// TIA Portal V21 program export: 7 tag tables, 1 data types, 19 data blocks, 22 code blocks (in call order from the OBs), 253 instance data blocks

VAR_GLOBAL   // PLC tag table "ALARM BIT"
   "DOOR1 CLOSE PB BIT" AT %M145.0 : Bool;
   "PV BOILER TEMP" AT %MD146 : Real;
   "SET BOILER BIT" AT %M145.1 : Bool;
   "PLANT STEAM LOW BIT" AT %M145.2 : Bool;
   "PURE STEAM LOW BIT" AT %M145.3 : Bool;
   "COOLING WATER LOW BIT" AT %M145.4 : Bool;
   "DOOR1 SAFETY SENSOR BIT" AT %M145.5 : Bool;
   "DOOR2 SAFETY SENSOR BIT" AT %M145.6 : Bool;
   "BOILER WATER OK BIT" AT %M145.7 : Bool;
   "RESET C21" AT %M152.2 : Bool;
   "MAN BOILER INLET VAL" AT %M152.3 : Bool;
   RESET_c22 AT %M152.4 : Bool;
   PULSE63 AT %M152.5 : Bool;
   PULSE64 AT %M152.6 : Bool;
   "door2 allow" AT %M152.7 : Bool;
   Cham_exh_val_bit AT %M160.0 : Bool;
   pulse65 AT %M160.1 : Bool;
   "abort standard" AT %M160.2 : Bool;
   PULSE66 AT %M154.0 : Bool;
END_VAR

VAR_GLOBAL   // PLC tag table "ANALOG"
   "DOOR1 PRESSURE" AT %IW120 : Int;
   "DOOR2 PRESSURE" AT %IW122 : Int;
   "JACKET PRESSURE" AT %IW124 : Int;
   "CHAMBER PRESSURE" AT %IW126 : Int;
END_VAR

VAR_GLOBAL   // PLC tag table "BIT"
END_VAR

VAR_GLOBAL   // PLC tag table "DI"
   "EMG SWITCH" AT %I0.0 : Bool;
   "RESET PB" AT %I0.1 : Bool;
   "VACUUM PUMP TRIP" AT %I0.2 : Bool;
   "DOOR1 OPEN LMT" AT %I0.3 : Bool;
   "DOOR1 CLOSE LMT" AT %I0.4 : Bool;
   "DOOR2 OPEN LMT" AT %I0.5 : Bool;
   "DOOR2 CLOSE LMT" AT %I0.6 : Bool;
   "DOOR2 CLOSE PB" AT %I0.7 : Bool;
   "DOOR2 OPEN PB" AT %I1.0 : Bool;
   "DOOR1 CLOSE PB" AT %I1.1 : Bool;
   "DOOR1 OPEN PB" AT %I1.2 : Bool;
   "AIR PREESURE SWS" AT %I1.3 : Bool;
   "plant steam low" AT %I1.4 : Bool;
   "pure steam low" AT %I1.5 : Bool;
   "cooling wtr low" AT %I2.0 : Bool;
   SPP AT %I2.1 : Bool;
   "DOOR1 CURTAIN SENSOR" AT %I2.2 : Bool;
   "DOOR2 CURTAIN SENSOR" AT %I2.3 : Bool;
   "BOILER WATER LEVEL OK" AT %I2.4 : Bool;
   "DRUM VFD TRIP" AT %I10.2 : Bool;
   "CRC PUMP TRIP" AT %I10.4 : Bool;
END_VAR

VAR_GLOBAL   // PLC tag table "DO"
   "VCC PUMP" AT %Q0.0 : Bool;   // VCC PUMP
   "DOOR1 GASKET" AT %Q0.1 : Bool;   // DOOR1 GASKET
   "DOOR1 VCC" AT %Q0.2 : Bool;   // DOOR1 VCC
   "DOOR2 GASKET" AT %Q0.3 : Bool;   // DOOR2 GASKET
   "DOOR2 VCC" AT %Q0.4 : Bool;   // DOOR2 VCC
   "JACKET STEAM VAL" AT %Q0.5 : Bool;   // JACKET STEAM VAL
   "JACKET STEAM OUT" AT %Q0.6 : Bool;
   "CHAMBER STEAM VAL" AT %Q0.7 : Bool;   // CHAMBER STEAM VAL
   "CHAMBER STEAM SMALL" AT %Q1.0 : Bool;   // DOOR2 INTERLOCK VAL
   "CHAMBER EXHAUST VAL" AT %Q1.1 : Bool;   // CHAMBER EXHAUST VAL
   "DRAIN VAL" AT %Q2.0 : Bool;   // DRAIN VAL
   "CHAMBER VACCUM VAL" AT %Q2.1 : Bool;
   "CHAMBER VENT VAL" AT %Q2.2 : Bool;   // CHAMBER VENT VAL
   "DOOR1 OPEN VAL" AT %Q2.3 : Bool;   // DOOR1 OPEN VAL
   "DOOR1 CLOSE VAL" AT %Q2.4 : Bool;   // DOOR1 CLOSE VAL
   "DOOR2 OPEN VAL" AT %Q2.5 : Bool;   // DOOR2 OPEN VAL
   "DOOR2 CLOSE VAL" AT %Q2.6 : Bool;   // DOOR2 CLOSE VAL
   "PROCESS ON IND" AT %Q2.7 : Bool;   // WFI VAL
   "door1 precondition lamp" AT %Q3.0 : Bool;
   "door2 precondition lamp" AT %Q3.1 : Bool;
   "DOOR1 OPEN LAMP" AT %Q3.2 : Bool;   // PWD VAL
   "DOOR2 OPEN LAMP" AT %Q3.3 : Bool;   // PWD CRC VAL
   HOOTER AT %Q3.4 : Bool;   // HOOTER
   "CHAMBER CONDENSOR VAL" AT %Q3.5 : Bool;   // CHAMBER CONDENSOR VAL
   "BOILER HEATER" AT %Q3.6 : Bool;   // BOILER HEATER
   "CRC MOTOR" AT %Q10.2 : Bool;   // CRC MOTOR
   "DETERGENT DSG VAL" AT %Q12.2 : Bool;   // DETERGENT DSG VAL
   "SILICON DSG VAL" AT %Q12.3 : Bool;   // SILICON DSG VAL
   "CHAMBER AIR VENT FAST" AT %Q18.6 : Bool;   // DOOR1 INTERLOCK VAL
END_VAR

VAR_GLOBAL   // PLC tag table "Default tag table"
   "REC DOOR1 PRESSURE" AT %QW150 : Int;
   "REC DOOR2 PRESSURE" AT %QW152 : Int;
   "REC CHAMBER PRESSURE" AT %QW154 : Int;
   "REC JACKET PRESSURE" AT %QW156 : Int;
   "REC DRUM SPEED" AT %QW158 : Int;
   "PRINT START" AT %M0.0 : Bool;
   TRIGGER AT %M0.1 : Bool;
   LENGTH AT %MW2 : Int;
   "NOT" AT %M0.2 : Bool;
   HIT AT %M0.3 : Bool;
   "START PV" AT %M0.4 : Bool;
   Clock_Byte AT %MB500 : Byte;
   Clock_10Hz AT %M500.0 : Bool;
   Clock_5Hz AT %M500.1 : Bool;
   "Clock_2.5Hz" AT %M500.2 : Bool;
   Clock_2Hz AT %M500.3 : Bool;
   "Clock_1.25Hz" AT %M500.4 : Bool;
   Clock_1Hz AT %M500.5 : Bool;
   "Clock_0.625Hz" AT %M500.6 : Bool;
   "Clock_0.5Hz" AT %M500.7 : Bool;
   System_Byte AT %MB1 : Byte;
   FirstScan AT %M1.0 : Bool;
   DiagStatusUpdate AT %M1.1 : Bool;
   AlwaysTRUE AT %M1.2 : Bool;
   AlwaysFALSE AT %M1.3 : Bool;
   AHJGSJH AT %MB4 : Byte;
   JGJH AT %MB5 : Byte;
   GET_DAY AT %MB180 : Byte;
   GET_MONTH AT %MB181 : Byte;
   GET_YEAR AT %MB182 : Byte;
   DAY AT %MW32 : Int;
   MONTH AT %MW44 : Int;
   YEAR AT %MW10 : Int;
   GET_HOUR AT %MB183 : Byte;
   GET_MINUTE AT %MB184 : Byte;
   GET_SECOND AT %MB185 : Byte;
   HOUR AT %MW40 : Int;
   MINUTE AT %MW42 : Int;
   SECOND AT %MW12 : Int;
   "NILESH BHAU" AT %MB6 : Byte;
   GET_CONTROL_TEMP AT %MD1400 : Real;
   "SP_CONTROL TEMP" AT %MD60 : Real;
   GET_CONVEYOR_SPEED AT %MD1404 : Real;
   SP_CONVEYOR_SPEED AT %MD64 : Real;
   "DRY ZONE REAL" AT %MD16 : Real;
   "GET_CONVEYOR ON TEMP" AT %MD1408 : Real;
   SP_CONVEYOR_ON_TEMP AT %MD68 : Real;
   "GET_CONVEYOR OFF TEMP" AT %MD1412 : Real;
   SP_CONVEYOR_OFF_TEMP AT %MD72 : Real;
   GET_DZ_PV AT %MD1416 : Real;
   DZ_PV AT %MD20 : Real;
   GET_MHZ_PV AT %MD1420 : Real;
   MHZ_PV AT %MD76 : Real;
   GET_STR_IN_PV AT %MD1424 : Real;
   STR_IN_PV AT %MD24 : Real;
   GET_STR_OUT_PV AT %MD1428 : Real;
   STR_OUT_PV AT %MD80 : Real;
   GET_CLZ_UP_PV AT %MD1432 : Real;
   CLZ_UP_PV AT %MD84 : Real;
   GET_CLZ_DWN_PV AT %MD1436 : Real;
   CLZ_DWN_PV AT %MD28 : Real;
   "GET_CONVEYOR SPEED_PV" AT %MD1440 : Real;
   "CONVEYOR SPEED_PV" AT %MD36 : Real;
   KJAHKJH AT %MD46 : Real;
   GET_MODE AT %MB197 : Byte;
   MODE AT %MW14 : Int;
   GET_PROCESS_HOUR AT %MB198 : Byte;
   PROCESS_HOUR AT %MW50 : Int;
   GET_PROCESS_MINUTE AT %MB199 : Byte;
   PROCESS_MINUTE AT %MW52 : Int;
   GET_PROCESS_SEC AT %MB200 : Byte;
   PROCESS_SEC AT %MW54 : Int;
   AL1 AT %M115.0 : Bool;
   "AL EMG STOP" AT %M115.1 : Bool;
   "AL DRUM TRIP" AT %M115.2 : Bool;
   "AL VACUUM TRIP" AT %M115.3 : Bool;
   "AL CRC TRIP" AT %M115.4 : Bool;
   AL6 AT %M115.5 : Bool;
   AL7 AT %M115.6 : Bool;
   AL8 AT %M115.7 : Bool;
   AL9 AT %M114.0 : Bool;
   AL10 AT %M114.1 : Bool;
   AL11 AT %M114.2 : Bool;
   AL12 AT %M114.3 : Bool;
   "AL JACKET RTD FAIL" AT %M114.4 : Bool;
   "AL CHAM RTD FAIL" AT %M114.5 : Bool;
   "AL AIR FAIL" AT %M114.6 : Bool;
   AL16 AT %M114.7 : Bool;
   AL1_1 AT %M118.0 : Bool;
   AL1_2 AT %M118.1 : Bool;
   AL1_3 AT %M118.2 : Bool;
   "AL JACKET PRESS FAIL" AT %M118.3 : Bool;
   "AL DOOR1 PRESS FAIL" AT %M118.4 : Bool;
   "AL DOOR2 PRESS FAIL" AT %M118.5 : Bool;
   "AL CHAM PRESS FAIL" AT %M118.6 : Bool;
   AL1_8 AT %M118.7 : Bool;
   "AL DOOR1 CL LMT FAIL" AT %M117.0 : Bool;
   AL2_10 AT %M117.1 : Bool;
   AL2_11 AT %M117.2 : Bool;
   AL2_12 AT %M117.3 : Bool;
   "AL DOOR2 CL LMT FAIL" AT %M117.4 : Bool;
   AL2_14 AT %M117.5 : Bool;
   AL2_15 AT %M117.6 : Bool;
   AL2_16 AT %M117.7 : Bool;
   "REQ AL1" AT %M0.5 : Bool;
   "AL1 TRIG" AT %M0.6 : Bool;
   "REQ AL3" AT %M0.7 : Bool;
   "AL3 TRIG" AT %M7.0 : Bool;
   "REQ AL4" AT %M7.1 : Bool;
   "AL4 TRIG" AT %M7.2 : Bool;
   "AL5 TRIG" AT %M7.3 : Bool;
   "REQ AL5" AT %M7.4 : Bool;
   "AL6 TRIG" AT %M7.5 : Bool;
   "REQ AL6" AT %M7.6 : Bool;
   "AL7 TRIG" AT %M7.7 : Bool;
   "REQ AL7" AT %M56.0 : Bool;
   "AL8 TRIG" AT %M56.1 : Bool;
   "REQ AL8" AT %M56.2 : Bool;
   "AL11 TRIG" AT %M56.3 : Bool;
   "REQ AL11" AT %M56.4 : Bool;
   "AL12 TRIG" AT %M56.5 : Bool;
   "REQ AL12" AT %M56.6 : Bool;
   "AL14 TRIG" AT %M56.7 : Bool;
   "REQ AL14" AT %M57.0 : Bool;
   "AL1_1 TRIG" AT %M57.1 : Bool;
   "REQ AL1_1" AT %M57.2 : Bool;
   "AL1_3 TRIG" AT %M57.3 : Bool;
   "REQ AL1_3" AT %M57.4 : Bool;
   "AL1_5 TRIG" AT %M57.5 : Bool;
   "REQ AL1_5" AT %M57.6 : Bool;
   "AL1_6 TRIG" AT %M57.7 : Bool;
   "REQ AL1_6" AT %M58.0 : Bool;
   "AL1_7 TRIG" AT %M58.1 : Bool;
   "REQ AL1_7" AT %M58.2 : Bool;
   "AL1_8 TRIG" AT %M58.3 : Bool;
   "REQ AL1_8" AT %M58.4 : Bool;
   "AL2_9 TRIG" AT %M58.5 : Bool;
   "REQ AL2_9" AT %M58.6 : Bool;
   "AL2_14 TRIG" AT %M58.7 : Bool;
   "REQ AL2_14" AT %M59.0 : Bool;
   "EMG SEL BIT" AT %M8.0 : Bool;
   "PHASE FAIL SEL BIT" AT %M8.1 : Bool;
   "COVEYOR SEL BIT" AT %M8.2 : Bool;
   "HEATER SEL BIT" AT %M8.3 : Bool;
   "TEMP SEL BIT" AT %M8.4 : Bool;
   "DRY ZONE SEL BIT" AT %M8.5 : Bool;
   "COOL ZONE SEL BIT" AT %M8.6 : Bool;
   "STR ZONE BIT" AT %M8.7 : Bool;
   "VAPOR TRIP SEL BIT" AT %M9.0 : Bool;
   "TURBINE TRIP SEL BIT" AT %M9.1 : Bool;
   "VAPOR SUPPLY SEL BIT" AT %M9.2 : Bool;
   "CONV OVER SEL BIT" AT %M9.3 : Bool;
   "LAF FAIL SEL BIT" AT %M9.4 : Bool;
   "GET_SHUDOWN BUFF" AT %MW1444 : Int;
   "SHUDOWN BUFF" AT %MW34 : Int;
   SHUT AT %M9.5 : Bool;
   "REQ SHUT" AT %M9.6 : Bool;
   LAST AT %MB1446 : Byte;
   "LAST TRIG" AT %M9.7 : Bool;
   OVER AT %M59.1 : Bool;
   "P OVER" AT %M59.2 : Bool;
   "PRINT STOP" AT %M59.3 : Bool;
   "PRINT STOP TRIG" AT %M59.4 : Bool;
   "HEAT UP 1 ON" AT %M59.5 : Bool;
   "HEAT UP 2 ON" AT %M59.6 : Bool;
   "HEAT UP 3 ON" AT %M59.7 : Bool;
   "HEAT UP 4 ON" AT %M88.0 : Bool;
   "CONV TEMP ON" AT %M88.1 : Bool;
   "V HIGH PRESS" AT %M151.0 : Bool;
   "AL DOOR2 OP LMT FAIL" AT %M151.1 : Bool;
   "AL DOOR1 OP LMT FAIL" AT %M151.2 : Bool;
   "AL STER_TIME_STOP" AT %M700.0 : Bool;
   "AL TURB SUP FAIL" AT %M151.4 : Bool;
   "AL STER_HOLD TIME RESET" AT %M151.5 : Bool;
   "AL HEATER SUP FAIL" AT %M151.6 : Bool;
   "AL_JACKET HEATING FAIL" AT %M151.7 : Bool;
   "AL_STER_HOLD HEATING FAIL" AT %M150.0 : Bool;
   AL_TOO_LATE_VACUUM AT %M150.1 : Bool;
   "AL BOILER WATER LOW" AT %M150.2 : Bool;
   "AL_DOOR1 SAFETY SENSOR FAIL" AT %M150.3 : Bool;
   "AL PHASE FAIL" AT %M150.4 : Bool;
   "1ML OK" AT %M88.2 : Bool;
   "2ML OK" AT %M88.3 : Bool;
   "3ML OK" AT %M88.4 : Bool;
   "5ML OK" AT %M88.5 : Bool;
   "10ML OK" AT %M88.6 : Bool;
   "HOOTER RESET BIT" AT %M88.7 : Bool;
   "CON ANNI" AT %M89.0 : Bool;
   "MANUAL INFEED" AT %M89.1 : Bool;
   "VPR ANN" AT %M89.2 : Bool;
   "LAF ANN" AT %M89.3 : Bool;
   "100ML OK" AT %M89.4 : Bool;
   "TURBINE SUP SEL BIT" AT %M89.5 : Bool;
   "AL VACUUM BREAK FAIL" AT %M150.6 : Bool;
   "AL DOOR PRECOND FAIL" AT %M150.7 : Bool;
   "AL JACKET PRESSURE HH" AT %M153.0 : Bool;
   BL1 AT %MW90 : Int;
   "AL DRY ZONE HIGH" AT %M153.2 : Bool;
   RESET AT %M89.6 : Bool;
   "LAF ON" AT %M89.7 : Bool;
   OFF AT %M92.0 : Bool;
   "VPR ON" AT %M92.1 : Bool;
   OFF1 AT %M92.2 : Bool;
   "TURB ON" AT %M92.3 : Bool;
   OFF2 AT %M92.4 : Bool;
   "HEAT ON" AT %M92.5 : Bool;
   OFF3 AT %M92.6 : Bool;
   "CONV ON" AT %M92.7 : Bool;
   "OFF 4" AT %M93.0 : Bool;
   "DOWNLOAD RC" AT %M93.1 : Bool;
   "AL HOT PRS LOW" AT %M153.1 : Bool;
   "AL COOL PRS HIGH" AT %M153.3 : Bool;
   Tag_1 AT %M153.4 : Bool;
   "AL CONV OVER" AT %M153.5 : Bool;
   "AL LAF PRESS SWS" AT %M153.6 : Bool;
   "HEATER 2" AT %M93.2 : Bool;
   OFFF AT %M93.3 : Bool;
   "HEATER 3" AT %M93.4 : Bool;
   OFFF1 AT %M93.5 : Bool;
   "HEATER 4" AT %M93.6 : Bool;
   OFFF44 AT %M93.7 : Bool;
   Tag_3 AT %M153.7 : Bool;
   Tag_4 AT %M152.0 : Bool;
   "CONVEYOR TRIP SEL BIT" AT %M110.0 : Bool;
   OFFFFFF AT %M94.0 : Bool;
   "PRINT SPEED" AT %MD96 : Real;
   TURBINE2 AT %M94.1 : Bool;
   OK AT %M94.2 : Bool;
   RESETC1 AT %M94.3 : Bool;
   POPUP AT %M152.1 : Bool;
   RESETC3 AT %M94.4 : Bool;
   RESETC4 AT %M94.5 : Bool;
   RESETC5 AT %M94.6 : Bool;
   RESETC6 AT %M94.7 : Bool;
   RESETC7 AT %M95.0 : Bool;
   RESETC8 AT %M95.1 : Bool;
   RESETC9 AT %M95.2 : Bool;
   RESETC10 AT %M95.3 : Bool;
   RESETC11 AT %M95.4 : Bool;
   RESETT5 AT %M95.5 : Bool;
   RESETC12 AT %M95.6 : Bool;
   RESETT6 AT %M95.7 : Bool;
   RESETC13 AT %M100.0 : Bool;
   RESETT7 AT %M100.1 : Bool;
   RESETC14 AT %M100.2 : Bool;
   RESETT8 AT %M100.3 : Bool;
   RESETC15 AT %M100.4 : Bool;
   RESETC16 AT %M100.5 : Bool;
   RESETC17 AT %M100.6 : Bool;
   RESETC18 AT %M100.7 : Bool;
   RESETT12 AT %M101.0 : Bool;
   RESETC19 AT %M101.1 : Bool;
   RESETC20 AT %M101.2 : Bool;
   RESETC21 AT %M101.3 : Bool;
   RESETC22 AT %M101.4 : Bool;
   RESETT16 AT %M101.5 : Bool;
   RESETC23 AT %M101.6 : Bool;
   RESETC24 AT %M101.7 : Bool;
   RESETC25 AT %M102.0 : Bool;
   RESETC26 AT %M102.1 : Bool;
   RESETC27 AT %M102.2 : Bool;
   RESETT21 AT %M102.3 : Bool;
   RESETC28 AT %M102.4 : Bool;
   RESETT22 AT %M102.5 : Bool;
   RESETC29 AT %M102.6 : Bool;
   RESETT23 AT %M102.7 : Bool;
   RESETC30 AT %M103.0 : Bool;
   "DRUM MOTOR BIT" AT %M103.1 : Bool;
   "EXH ON" AT %M103.2 : Bool;
   RESETC32 AT %M103.3 : Bool;
   "CONTROL CHMB" AT %M103.4 : Bool;
   "STERILE TEMP ON" AT %MD104 : Real;
   "PWD TEMP ON" AT %MD120 : Real;
   resetc33 AT %M103.5 : Bool;
   "vaccum ok" AT %M103.6 : Bool;
   trigger2 AT %M103.7 : Bool;
   "VCC DIFF" AT %MD124 : Real;
   LENGTH2 AT %MW108 : Int;
   "CYCLE END" AT %M110.1 : Bool;
   ERROR AT %M110.2 : Bool;
   "RESET HPHV VCC" AT %M110.3 : Bool;
   "RESETBOW VCC" AT %M110.4 : Bool;
   okkk AT %M110.5 : Bool;
   "one shot" AT %M110.6 : Bool;
   "jack out set" AT %M110.7 : Bool;
   resetct3 AT %M111.0 : Bool;
   resetct4 AT %M111.1 : Bool;
   "hphv ok" AT %M111.2 : Bool;
   "bowie ok" AT %M111.3 : Bool;
   "std ok" AT %M111.4 : Bool;
   sterileok AT %M111.5 : Bool;
   "TEST BIT" AT %M111.6 : Bool;
   "TEST BIT2" AT %M111.7 : Bool;
   "CLOSURE ON" AT %M112.0 : Bool;
   "CLOSE START" AT %M112.1 : Bool;
   "DEL LENGTH" AT %MW128 : Int;
   "RESET C5" AT %M112.2 : Bool;
   sip_ok AT %M112.3 : Bool;
   "sip ok1" AT %M112.4 : Bool;
   PULSE1 AT %M112.5 : Bool;
   PULSE2 AT %M112.6 : Bool;
   pulse3 AT %M112.7 : Bool;
   PP1 AT %M113.0 : Bool;
   PP2 AT %M113.1 : Bool;
   PP3 AT %M113.2 : Bool;
   PP4 AT %M113.3 : Bool;
   PP5 AT %M113.4 : Bool;
   pp6 AT %M113.5 : Bool;
   RESETCOUNT6 AT %M113.6 : Bool;
   RESETCOUNT7 AT %M113.7 : Bool;
   "VACCUM LEAK DIFF" AT %MD130 : Real;
   PULSE4 AT %M116.0 : Bool;
   PULSE5 AT %M116.1 : Bool;
   PULSE6 AT %M116.2 : Bool;
   PULSE7 AT %M116.3 : Bool;
   PULSE8 AT %M116.4 : Bool;
   PULSE9 AT %M116.5 : Bool;
   PULSE10 AT %M116.6 : Bool;
   PULSE11 AT %M116.7 : Bool;
   PULSE12 AT %M119.0 : Bool;
   PULSE13 AT %M119.1 : Bool;
   pulse14 AT %M119.2 : Bool;
   pulse15 AT %M119.3 : Bool;
   "STD1 SELECT" AT %M119.4 : Bool;
   "STD2 SELECT" AT %M119.5 : Bool;
   PULSE16 AT %M119.6 : Bool;
   PULSE17 AT %M119.7 : Bool;
   PULSE18 AT %M134.0 : Bool;
   PULSE19 AT %M134.1 : Bool;
   PULSE20 AT %M134.2 : Bool;
   pulse21 AT %M134.3 : Bool;
   "END PRINT OK" AT %M134.4 : Bool;
   PULSE22 AT %M134.5 : Bool;
   pulse23 AT %M134.6 : Bool;
   pulse24 AT %M134.7 : Bool;
   pulse25 AT %M135.0 : Bool;
   pulse26 AT %M135.1 : Bool;
   pulse27 AT %M135.2 : Bool;
   pulse28 AT %M135.3 : Bool;
   pulse29 AT %M135.4 : Bool;
   pulse30 AT %M135.5 : Bool;
   pulse31 AT %M135.6 : Bool;
   pulse32 AT %M135.7 : Bool;
   pulse33 AT %M136.0 : Bool;
   pulse34 AT %M136.1 : Bool;
   pulse35 AT %M136.2 : Bool;
   pulse36 AT %M136.3 : Bool;
   pulse37 AT %M136.4 : Bool;
   pulse38 AT %M136.5 : Bool;
   pulse39 AT %M136.6 : Bool;
   pulse40 AT %M136.7 : Bool;
   "start process" AT %M137.0 : Bool;
   PULSE41 AT %M137.1 : Bool;
   "START PROCES2" AT %M137.2 : Bool;
   PULSE42 AT %M137.3 : Bool;
   pulse43 AT %M137.4 : Bool;
   PULSE44 AT %M137.5 : Bool;
   PULSE45 AT %M137.6 : Bool;
   PULSE46 AT %M137.7 : Bool;
   PULSE47 AT %M138.0 : Bool;
   PULSE48 AT %M138.1 : Bool;
   PULSE49 AT %M138.2 : Bool;
   "hooter reset" AT %M138.3 : Bool;
   "RESET DOOR1" AT %M138.4 : Bool;
   "RESET DOOR2" AT %M138.5 : Bool;
   "STD3 SELECT" AT %M138.6 : Bool;
   "STD4 SELECT" AT %M138.7 : Bool;
   "STD5 SELECT" AT %M139.0 : Bool;
   "STD6 SELECT" AT %M139.1 : Bool;
   "STD7 SELECT" AT %M139.2 : Bool;
   "STD8 SELECT" AT %M139.3 : Bool;
   "STD9 SELECT" AT %M139.4 : Bool;
   "VACCUM FAIL" AT %M139.5 : Bool;
   "hold start" AT %M139.6 : Bool;
   RESETT169 AT %M139.7 : Bool;
   RESET_C8 AT %M140.0 : Bool;
   RESETT171 AT %M140.1 : Bool;
   RESETC_9 AT %M140.2 : Bool;
   RESETT174 AT %M140.3 : Bool;
   RESET_C10 AT %M140.4 : Bool;
   RESETT177 AT %M140.5 : Bool;
   RESET_C11 AT %M140.6 : Bool;
   RESETT179 AT %M140.7 : Bool;
   RESET_C12 AT %M141.0 : Bool;
   RESETT184 AT %M141.1 : Bool;
   RESET_C13 AT %M141.2 : Bool;
   RESETT185 AT %M141.3 : Bool;
   RESET_C14 AT %M141.4 : Bool;
   RESET_C15 AT %M141.5 : Bool;
   "RESET C16" AT %M141.6 : Bool;
   "RESET C17" AT %M141.7 : Bool;
   "reset c18" AT %M142.0 : Bool;
   RESET_C19 AT %M142.1 : Bool;
   "STANDARD DONE" AT %M142.2 : Bool;
   "HPHV DONE" AT %M142.3 : Bool;
   "BOW DONE" AT %M142.4 : Bool;
   "VACUUM DONE" AT %M142.5 : Bool;
   PULSE50 AT %M142.6 : Bool;
   "RESET C7" AT %M142.7 : Bool;
   pulse51 AT %M143.0 : Bool;
   pulse52 AT %M143.1 : Bool;
   Tag_2 AT %M151.3 : Bool;
   "VLT OG" AT %M143.2 : Bool;
   "VLT EX" AT %M143.3 : Bool;
   AMP_VLT AT %M143.4 : Bool;
   "CYCLE STOP PRESS" AT %M143.5 : Bool;
   PULSE53 AT %M143.6 : Bool;
   "STER HEAT AGAIN" AT %M143.7 : Bool;
   "STER HEAT FAIL" AT %M144.0 : Bool;
   PULSE54 AT %M144.1 : Bool;
   PULSE55 AT %M144.2 : Bool;
   reset_c20 AT %M144.3 : Bool;
   PULSE60 AT %M144.4 : Bool;
   PULSE61 AT %M144.5 : Bool;
   PULSE62 AT %M144.6 : Bool;
   PULSE56 AT %M144.7 : Bool;
   "AL_DOOR2 SAFETY SENSOR FAIL" AT %M150.5 : Bool;
   "BOILER WATER INLET VAL" AT %Q3.7 : Bool;
END_VAR

VAR_GLOBAL   // PLC tag table "RTD"
   "CHAMBER DRAIN TEMP" AT %IW100 : Int;
   "CHAMBER TEMP1" AT %IW102 : Int;
   "CHAMBER TEMP2" AT %IW104 : Int;
   "CHAMBER TEMP3" AT %IW106 : Int;
   "CHAMBER TEMP4" AT %IW108 : Int;
   "JACKET TEMP" AT %IW110 : Int;
END_VAR

TYPE "STD"
   STRUCT
      "SET TEMP1" : Real := 0.0;
      "SET TEMP2" : Real := 0.0;
      "SET TEMP3" : Real := 0.0;
      "SET PRESS" : Real := 0.0;
      "SET HOLD1" : Int := 0;
      "SET HOLD2" : Int := 0;
      "SET HOLD3" : Int := 0;
      "SET VCC" : Real := 0.0;
      "SET UP PRESS" : Real := 0.0;
      "SET VCC HOLD" : Int := 0;
      "SET NO OF PULSE" : Int := 0;
   END_STRUCT;
END_TYPE

DATA_BLOCK "ADD_ON"   // DB263
{ S7_Optimized_Access := 'FALSE' }
   VAR RETAIN
      "SET TEMP1 STD3" : Real := 100.0;
      "SET TEMP2 STD3" : Real := 110.0;
      "SET TEMP3 STD3" : Real := 121.4;
      "SET PRESS STD3" : Real := 0.05;
      "SET HOLD1 STD3" : Int := 5;
      "SET HOLD2 STD3" : Int := 5;
      "SET HOLD3 STD3" : Int := 30;
      "SET VCC STD3" : Real := 0.0;
      "SET UP PRESS STD3" : Real := 0.0;
      "SET VCC HOLD STD3" : Int := 0;
      "SET NO OF PULSE STD3" : Int := 0;
      "SET TEMP1 STD4" : Real := 100.0;
      "SET TEMP2 STD4" : Real := 110.0;
      "SET TEMP3 STD4" : Real := 121.4;
      "SET PRESS STD4" : Real := 0.05;
      "SET HOLD1 STD4" : Int := 5;
      "SET HOLD2 STD4" : Int := 5;
      "SET HOLD3 STD4" : Int := 30;
      "SET VCC STD4" : Real := 0.0;
      "SET UP PRESS STD4" : Real := 0.0;
      "SET VCC HOLD STD4" : Int := 0;
      "SET NO OF PULSE STD4" : Int := 0;
      "SET TEMP1 STD5" : Real := 100.0;
      "SET TEMP2 STD5" : Real := 110.0;
      "SET TEMP3 STD5" : Real := 121.4;
      "SET PRESS STD5" : Real := 0.05;
      "SET HOLD1 STD5" : Int := 5;
      "SET HOLD2 STD5" : Int := 5;
      "SET HOLD3 STD5" : Int := 30;
      "SET VCC STD5" : Real := 0.0;
      "SET UP PRESS STD5" : Real := 0.0;
      "SET VCC HOLD STD5" : Int := 0;
      "SET NO OF PULSE STD5" : Int := 0;
      "SET TEMP1 STD6" : Real := 100.0;
      "SET TEMP2 STD6" : Real := 110.0;
      "SET TEMP3 STD6" : Real := 121.4;
      "SET PRESS STD6" : Real := 0.05;
      "SET HOLD1 STD6" : Int := 5;
      "SET HOLD2 STD6" : Int := 5;
      "SET HOLD3 STD6" : Int := 30;
      "SET VCC STD6" : Real := 0.0;
      "SET UP PRESS STD6" : Real := 0.0;
      "SET VCC HOLD STD6" : Int := 0;
      "SET NO OF PULSE STD6" : Int := 0;
      "SET TEMP1 STD7" : Real := 100.0;
      "SET TEMP2 STD7" : Real := 110.0;
      "SET TEMP3 STD7" : Real := 121.4;
      "SET PRESS STD7" : Real := 0.05;
      "SET HOLD1 STD7" : Int := 5;
      "SET HOLD2 STD7" : Int := 5;
      "SET HOLD3 STD7" : Int := 30;
      "SET VCC STD7" : Real := 0.0;
      "SET UP PRESS STD7" : Real := 0.0;
      "SET VCC HOLD STD7" : Int := 0;
      "SET NO OF PULSE STD7" : Int := 0;
      "SET TEMP1 STD8" : Real := 100.0;
      "SET TEMP2 STD8" : Real := 110.0;
      "SET TEMP3 STD8" : Real := 121.4;
      "SET PRESS STD8" : Real := 0.05;
      "SET HOLD1 STD8" : Int := 5;
      "SET HOLD2 STD8" : Int := 5;
      "SET HOLD3 STD8" : Int := 30;
      "SET VCC STD8" : Real := 0.0;
      "SET UP PRESS STD8" : Real := 0.0;
      "SET VCC HOLD STD8" : Int := 0;
      "SET NO OF PULSE STD8" : Int := 0;
      "SET TEMP1 STD9" : Real := 100.0;
      "SET TEMP2 STD9" : Real := 110.0;
      "SET TEMP3 STD9" : Real := 121.4;
      "SET PRESS STD9" : Real := 0.05;
      "SET HOLD1 STD9" : Int := 5;
      "SET HOLD2 STD9" : Int := 5;
      "SET HOLD3 STD9" : Int := 30;
      "SET VCC STD9" : Real := 0.0;
      "SET UP PRESS STD9" : Real := 0.0;
      "SET VCC HOLD STD9" : Int := 0;
      "SET NO OF PULSE STD9" : Int := 0;
      "SET LEAK VCC" : Real := -0.7;
      "SET VCC PRESS" : Real := -0.05;
      "SET DELAY BEFORE HOLD TIME" : Int := 0;
      "SET VCC HOLD TIME" : Int := 10;
      "SET ACCEPTANCE LEAK" : Real := 0.013;
   END_VAR
BEGIN
END_DATA_BLOCK

DATA_BLOCK "ALARM"   // DB101
{ S7_Optimized_Access := 'FALSE' }
   VAR
      AL_EMG_STOP : Bool;
      AL_LOW_PRESSURE : Bool;
      AL_DOOR_OPEN : Bool;
      AL_DRUM_MTR_TRIP : Bool;
      AL_VACCUM_MTR_TRIP : Bool;
      AL_RECRC_TRIP : Bool;
      AL_PW_START : Bool;
      AL_PW_OVER : Bool;
      AL_WFI_START : Bool;
      AL_WFI_OVER : Bool;
      AL_STERILE_START : Bool;
      AL_STERILE_OVER : Bool;
      AL_DRY_START : Bool;
      AL_DRY_OVER : Bool;
      AL_PROCESS_COMP : Bool;
      AL_PRESSURE_HIGH : Bool;
      AL_RTD_FAIL : Bool;
      "AL_CHAMBER PRESS_FAIL" : Bool;
      "AL DOOR1 CLOSE LMT FAIL" : Bool;
      "AL DOOR2 CLOSE LMT FAIL" : Bool;
      "AL CHAMBER PRESS HIGH" : Bool;
      "AL JACKET RTD FAIL" : Bool;
      "AL BOILER TEMP HIGH" : Bool;
      "AL DOOR1 VCC FAIL" : Bool;
      "AL DOOR2 VCC FAIL" : Bool;
      "AL PHASE FAILURE" : Bool;
      "AL TEMP OVERSHOOT" : Bool;
      "AL CHAMBER RTD1 FAIL" : Bool;
      "AL CHAMBER RTD2 FAIL" : Bool;
      "AL CHAMBER RTD3 FAIL" : Bool;
      "AL CHAMBER RTD4 FAIL" : Bool;
      "AL JACKET PRESS FAIL" : Bool;
      "AL DOOR1 PRESS FAIL" : Bool;
      "AL DOOR2 PRESS FAIL" : Bool;
   END_VAR
BEGIN
END_DATA_BLOCK

DATA_BLOCK "AMEND"   // DB36
{ S7_Optimized_Access := 'FALSE' }
   VAR
      "PRODUCT NAME" : String[80] := '$L$RPRODUCT NAME        :';
      "BATCH NO" : String[80] := '$L$RBATCH NO            :';
      "OPERATOR NAME" : String[80] := '$L$ROPERATOR NAME       :UDAYLAL';
      "RECIPE TYPE" : String[80] := '$L$R        :';
      "EQUIPMENT ID" : String[80] := '$L$REQUIPMENT ID        :C1/A/INJ/AUT-05';
      "OP PRODUCT NAME" : String[80] := '';
      "TUNNEL MODE" : String[80] := '$L$RPROCESS                    :    NONE';
      CIP : String[30] := 'CLOSURE CYCLE SELECTED';
      STANDARD1 : String[30] := 'STANDARD1 CYCLE SELECTED';
      STANDARD2 : String[30] := 'STANDARD2 CYCLE SELECTED';
      BOWIE : String[30] := 'BOWIE DICK CYCLE SELECTED';
      NONE : String[30] := 'NONE';
      "BATCH SIZE" : String[80] := '  CYCLE NO            :0488';
      "CONTAINER SIZE" : String[80] := '  CONTAINER SIZE      :';
      HPHV : String[80] := 'HPHV CYCLE SELECTED';
      LEAK : String[80] := 'VACUUM LEAK TEST SELECTED';
      start : String[80] := '46';
      end : String[80] := '18:52:46';
      "END PV" : String[80] := '  18:52:46    0.086     48.4    103.2     92.2     93.1    105.8 ';
      "PRINT PV" : String[80] := '$L$R18:52:46    0.086     48.4    103.2     92.2     93.1    105.8  NOT START';
      "PRINT CYCLE ABORT" : String[80] := '18:52:19   ******CYCLE ABORTED******     ';
      QUANTITY : String[80] := '  ';
   END_VAR
BEGIN
END_DATA_BLOCK

DATA_BLOCK "AUXILIARY"   // DB6
{ S7_Optimized_Access := 'TRUE' }
// stored: MemoryReserve 100
   VAR
      PULSE : Array[0..40] of Bool;
      "PWD STEAM ON" : Bool := TRUE;
      "CHAMBER TEMP" : Real := 0.0;
      "CHAMBER PRESS" : Real := 0.0;
      "START VACCUM" : Real := 0.0;
      "END VACCUM" : Real := 0.0;
      "ACTUAL LEAK" : Real := 0.0;
   END_VAR
   VAR RETAIN
      "STD TEMP1" : Real := 114.0;
      "STD TEMP2" : Real := 116.0;
      "STD TEMP3" : Real := 119.0;
      "STD PRESS" : Real := 0.1;
      "STD HOLD1" : Int := 5;
      "STD HOLD2" : Int := 3;
      "STD HOLD3" : Int := 2;
      "STD VCC" : Real := 0.0;
      "STD UP PRESS" : Real := 0.0;
      "STD VCC HOLD" : Int := 0;
      "NO OF STD PULSE" : Int := 0;
   END_VAR
   VAR
      "DRUM VFD" : Real := 8192.0;
      "STR STEAM ON" : Bool := FALSE;
      PULSE1 : Array[0..50] of Bool;
      pulse2 : Array[0..50] of Bool;
   END_VAR
   VAR RETAIN
      "STERILE HOLD TEMP" : Real := 121.4;
      "STERILE HOLD TIME" : Int := 30;
      "CONTROL BAND" : Real := 0.0;
      "STERILE STOP TEMP" : Real := 120.9;
   END_VAR
   VAR
      "STD CRITICAL TEMP" : Real;
   END_VAR
BEGIN
   PULSE[0..40] := FALSE;
   PULSE1[0..50] := FALSE;
   pulse2[0..50] := FALSE;
END_DATA_BLOCK

DATA_BLOCK "BUFF"   // DB82
{ S7_Optimized_Access := 'FALSE' }
   VAR
      MODE : Int;
      PROCESS : Int;
      DOOR1 : Int;
      DOOR2 : Int;
      SAFE : Int;
      "AUTO HMI" : Bool;
      "MANUAL HMI" : Bool;
      "STANDBY HMI" : Bool;
      "START HMI" : Bool;
      "STOP HMI" : Bool;
      SIP : Bool;
      STANDARD : Array[0..10] of Bool;
      STANDARD2 : Bool;
      "BOWIE DICK" : Bool;
      HPHV : Bool;
      "VCC LEAK" : Bool;
      DUMMY : Bool;
      DUMMY1 : Bool;
      "MAN VCC PUMP" : Bool;
      "MAN DOOR1 GASKET" : Bool;
      "MAN CRC MOTOR" : Bool;
      "MAN JACKET STEAM VAL" : Bool;
      "MAN CHAMBER STEAM VAL" : Bool;
      "MAN CHAMBER EXHAUST VAL" : Bool;
      "MAN CHAMBER VENT VAL" : Bool;
      "MAN CHAMBER CONDENSOR VAL" : Bool;
      "MAN WFI VAL" : Bool;
      "MAN PWD VAL" : Bool;
      "MAN PWD CRC VAL" : Bool;
      "MAN DETERGENT DSG VAL" : Bool;
      "MAN SILICON DSG VAL" : Bool;
      "MAN DRAIN VAL" : Bool;
      "MAN DOOR2 INTERLOCK VAL" : Bool;
      "MAN DOOR1 INTERLOCK VAL" : Bool;
      "MAN DOOR1 OPEN VAL" : Bool;
      "MAN DOOR1 CLOSE VAL" : Bool;
      "MAN DOOR2 OPEN VAL" : Bool;
      "MAN DOOR2 CLOSE VAL" : Bool;
      "MAN DOOR1 VCC" : Bool;
      "MAN DOOR2 GASKET" : Bool;
      "MAN DOOR2 VCC" : Bool;
      "MAN JACKET STEAM OUT" : Bool;
      "DOOR1 OPEN" : Bool;
      "DOOR1 CLOSE" : Bool;
      "DOOR2 OPEN" : Bool;
      "DOOR2 CLOSE" : Bool;
      "MAN DRUM MOTOR" : Bool;
      "MAN CHAMBER VACCUM VAL" : Bool;
      PRINT : Bool;
      "MAN CHAMBER STEAM SMALL" : Bool;
      "MAN CHAMBER AIR VENT" : Bool;
      "MAN JACKET STEAM OUT_1" : Bool;
      "MAN BOILER HEATER" : Bool;
   END_VAR
BEGIN
END_DATA_BLOCK

DATA_BLOCK "DATALOG"   // DB309
{ S7_Optimized_Access := 'FALSE' }
   VAR RETAIN
      "SET PRINT INTERVAL" : Int;
      "PROCESS PHASE" : Int;
      "TRIGGER BIT" : Bool;
      "START/STOP" : Bool;
      "BATCH DATA" : Struct
         "BATCH CODE" : WString;
         "BATCH NAME" : WString;
         "EQUIPMENT ID" : WString;
         "OPERATOR NAME" : WString;
         "PRODUCT NAME" : WString;
         "START DATE STRING" : WString;
         "END DATE STRING" : WString;
      END_STRUCT;
      INTERLOCK : Struct
         VACCUM : Struct
            START : Bool;
            STOP : Bool;
            NEW : Bool;
            BUFF : Int;
         END_STRUCT;
      END_STRUCT;
   END_VAR
BEGIN
END_DATA_BLOCK

DATA_BLOCK "DELTA D"   // DB183
{ S7_Optimized_Access := 'FALSE' }
   VAR
      TA : Real := 122.9;
      TB : Real := 121.0;
      Z : Real := 10.0;
      RATE : Real := 0.1900001;
      LEATHALTY : Real := 1.548817;
      "DELTA T" : Int := 15;
      F0 : Real := 13.06446;
      "MIN DRAIN" : Real := 51.8;
      "MAX DRAIN" : Real := 123.2;
      "MIN T1" : Real := 85.7;
      "MAX T1" : Real := 123.8;
      "MIN T2" : Real := 44.5;
      "MAX T2" : Real := 124.3;
      "MIN T3" : Real := 43.1;
      "MAX T3" : Real := 124.2;
      "MIN T4" : Real := 85.8;
      "MAX T4" : Real := 124.0;
      "MIN T5" : Real := 0.0;
      "MAX T5" : Real := 0.0;
      HEAD : String[80] := '$L$R                T1     T2     T3     T4      T5  ';   // 17,24,31,38,46
      "MIN TEMP" : String[80] := '$L$R  MIN TEMP  :                                                            ';   // 14
      "MAX TEMP" : String[80] := '$L$R  MAX TEMP  :                                                           ';   // 14
      "F ZERO" : String[80] := '$L$R  F0 VALUE  :                                                            ';   // 14
      "MIN F0" : String[80] := '$L$RTOTAL MINIMUM F0 VALUE ACHIEVED DURING CYLCE  :           ';   // 48
      "PRINT LINE" : String[80] := '   ';
      BIT : Array[0..10] of Bool;
      F1 : Real := 23.23226;
      F2 : Real := 27.93129;
      F3 : Real := 30.62606;
      F4 : Real := 30.62606;
      F5 : Real := 29.24768;
      "DEL TA" : Array[0..5] of Real;
      "DEL RATE" : Array[0..5] of Real;
      "DEL LEATH" : Array[0..5] of Real;
      dummy : Array[0..5] of Real;
   END_VAR
BEGIN
   BIT[0..10] := FALSE;
   "DEL TA"[0] := 123.7;
   "DEL TA"[1..2] := 124.1;
   "DEL TA"[3] := 123.9;
   "DEL TA"[4..5] := 0.0;
   "DEL RATE"[0] := 0.2699997;
   "DEL RATE"[1..2] := 0.3099999;
   "DEL RATE"[3] := 0.2900001;
   "DEL RATE"[4..5] := 0.0;
   "DEL LEATH"[0] := 1.862086;
   "DEL LEATH"[1..2] := 2.041737;
   "DEL LEATH"[3] := 1.949845;
   "DEL LEATH"[4..5] := 0.0;
END_DATA_BLOCK

DATA_BLOCK "DTL"   // DB100
{ S7_Optimized_Access := 'TRUE' }
// stored: MemoryReserve 100
   VAR RETAIN
      READ : DTL;
      WRITE : DTL;
      "RET READ" : Int := 0;
      "RET WRITE" : Int := 0;
      SET : Bool := FALSE;
   END_VAR
BEGIN
END_DATA_BLOCK

DATA_BLOCK "IO BITS"   // DB38
{ S7_Optimized_Access := 'TRUE' }
// stored: MemoryReserve 100
   VAR
      "DOOR1 PRESS BIT" : Bool;   // DOOR1 PRESS BIT
      "DOOR1 VCC BIT" : Bool;   // DOOR1 VCC BIT
      "DOOR2 VCC BIT" : Bool;   // DOOR2 VCC BIT
      "DOOR2 PRESS BIT" : Bool;   // DOOR2 PRESS BIT
      "JACKET SAFETY BIT" : Bool;   // JACKET SAFETY BIT
      "CHAMBER SAFETY BIT" : Bool;   // CHAMBER SAFETY BIT
      PFR : Bool;   // PFR
      "EMG SWITCH" : Bool;   // EMG SWITCH
      "RESET PB" : Bool;   // RESET PB
      "DRUM VFD TRIP" : Bool;   // DRUM VFD TRIP
      "VACCUM PUMP TRIP" : Bool;
      "CRC PUMP TRIP" : Bool;   // CRC PUMP TRIP
      "DOOR1 OPEN LMT" : Bool;   // DOOR1 OPEN LMT
      "DOOR1 CLOSE LMT" : Bool;   // DOOR1 CLOSE LMT
      "DOOR2 OPEN LMT" : Bool;   // DOOR2 OPEN LMT
      "DOOR2 CLOSE LMT" : Bool;   // DOOR2 CLOSE LMT
      "DOOR2 CLOSE PB" : Bool;   // DOOR2 CLOSE PB
      "DOOR2 OPEN PB" : Bool;   // DOOR2 OPEN PB
      "AIR PREESURE SWS" : Bool;   // AIR PREESURE SWS
      "I1.4 SPARE" : Bool;   // I1.4 SPARE
      "I1.5 SPARE" : Bool;   // I1.5 SPARE
      DUMMY : Bool;   // DUMMY
      DUMMY1 : Bool;   // DUMMY1
      "VCC PUMP" : Bool;   // VCC PUMP
      "DOOR1 GASKET" : Bool;   // DOOR1 GASKET
      "CRC MOTOR" : Bool;   // CRC MOTOR
      "JACKET STEAM VAL" : Bool;   // JACKET STEAM VAL
      "CHAMBER STEAM VAL" : Bool;   // CHAMBER STEAM VAL
      "CHAMBER EXHAUST VAL" : Bool;   // CHAMBER EXHAUST VAL
      "CHAMBER VENT VAL" : Bool;   // CHAMBER VENT VAL
      "CHAMBER CONDENSOR VAL" : Bool;   // CHAMBER CONDENSOR VAL
      "WFI VAL" : Bool;   // WFI VAL
      "PWD VAL" : Bool;   // PWD VAL
      "PWD CRC VAL" : Bool;   // PWD CRC VAL
      "DETERGENT DSG VAL" : Bool;   // DETERGENT DSG VAL
      "SILICON DSG VAL" : Bool;   // SILICON DSG VAL
      "DRAIN VAL" : Bool;   // DRAIN VAL
      "DOOR2 INTERLOCK VAL" : Bool;   // DOOR2 INTERLOCK VAL
      "DOOR1 INTERLOCK VAL" : Bool;   // DOOR1 INTERLOCK VAL
      "DOOR1 OPEN VAL" : Bool;   // DOOR1 OPEN VAL
      "DOOR1 CLOSE VAL" : Bool;   // DOOR1 CLOSE VAL
      "DOOR2 OPEN VAL" : Bool;   // DOOR2 OPEN VAL
      "DOOR2 CLOSE VAL" : Bool;   // DOOR2 CLOSE VAL
      "DOOR1 VCC" : Bool;   // DOOR1 VCC
      "DOOR2 GASKET" : Bool;   // DOOR2 GASKET
      "DOOR2 VCC" : Bool;   // DOOR2 VCC
      HOOTER : Bool;   // HOOTER
      "CHAMBER VACCUM VAL" : Bool;
      "CHAMBER STEAM SMALL VAL" : Bool;
      "CHAMBER AIR VENT FAST" : Bool;
      "JACKET STEAM OUT" : Bool;
      "BOW PULSE" : Array[0..100] of Bool;
      "HPHV PULSE" : Array[0..100] of Bool;
      "STANDARD PULSE" : Array[0..100] of Bool;
      "VACUUM PULSE" : Array[0..100] of Bool;
   END_VAR
BEGIN
END_DATA_BLOCK

DATA_BLOCK "L"   // DB187
{ S7_Optimized_Access := 'TRUE' }
// stored: MemoryReserve 100
   VAR RETAIN
      "DATE" : USInt;
      MONTH : USInt;
      YEAR : UInt;
      LO : Int;
      FIRMAWARE : Bool;
      "CIRON PRINT" : Bool;
      "STD VACUUM DIS" : Bool;
   END_VAR
BEGIN
END_DATA_BLOCK

DATA_BLOCK "MODBUS"   // DB99
{ S7_Optimized_Access := 'FALSE' }
   VAR
      "WRITE CONVEYOR" : Struct
         RUN : Int;
         SPEED : Int;
      END_STRUCT;
      "WRITE TURBINE" : Struct
         RUN : Int;
         SPEED : Int;
      END_STRUCT;
      "WRITE TURBINE2" : Struct
         RUN : Int;
         SPEED : Int;
      END_STRUCT;
      READ : Struct
         CONVEYOR : Int;
         TURBINE : Int;
         TURBINE2 : Int;
      END_STRUCT;
      "CONVEYOR STATUS" : Struct
         "W.DONE" : Bool;
         "W.ERROR" : Bool;
         "W.BUSY" : Bool;
         "W.STATUS" : Word;
         "R.DONE" : Bool;
         "R.ERROR" : Bool;
         "R.BUSY" : Bool;
         "R.STATUS" : Word;
      END_STRUCT;
      "TURBINE STATUS" : Struct
         "W.DONE" : Bool;
         "W.ERROR" : Bool;
         "W.BUSY" : Bool;
         "W.STATUS" : Word;
         "R.DONE" : Bool;
         "R.ERROR" : Bool;
         "R.BUSY" : Bool;
         "R.STATUS" : Word;
      END_STRUCT;
      "TURBINE2 STATUS" : Struct
         "W.DONE" : Bool;
         "W.ERROR" : Bool;
         "W.BUSY" : Bool;
         "W.STATUS" : Word;
         "R.DONE" : Bool;
         "R.ERROR" : Bool;
         "R.BUSY" : Bool;
         "R.STATUS" : Word;
      END_STRUCT;
      NOMX1 : Real;
      NOMX2 : Real;
      "NOM 3" : Real;
      "NOM 4" : Real;
      NOM5 : Real;
      NOM6 : Real;
      "READ TURB" : Struct
         "TURB1 READY" : Bool;
      END_STRUCT;
      "READ DRM" : Array[0..10] of Int;
   END_VAR
BEGIN
END_DATA_BLOCK

DATA_BLOCK "PI"   // DB144
{ S7_Optimized_Access := 'TRUE' }
// stored: MemoryReserve 100
   VAR
      NOM1 : Real;
      SETPOINT : Real;
      "PID OUT" : Real;
      NOM2 : Real;
      "PID IN" : Real;
   END_VAR
   VAR RETAIN
      GAIN : Real;
      "TIME" : Real;
   END_VAR
   VAR
      NOM3 : Real;
   END_VAR
BEGIN
END_DATA_BLOCK

DATA_BLOCK "PRINT DATA"   // DB39
{ S7_Optimized_Access := 'FALSE' }
   VAR RETAIN
      "PRINT INTERVAL" : Int := 0;
      "PRODUCT NAME" : String := '';
      "BATCH NO" : String := '';
      "OPERATOR NAME" : String := 'UDAYLAL';
      "RECIPE TYPE" : String := '  ';
      "EQUIPMENT ID" : String := 'C1/A/INJ/AUT-05';
      "TUNNEL MODE" : String := 'STANDARD3 CYCLE SELECTED';
      "BATCH SIZE" : String := '0488';
      "CONTAINER NO" : String := '';
      NEW : String := '';
      QUANTITY : String;
   END_VAR
BEGIN
END_DATA_BLOCK

DATA_BLOCK "PRINTING_1"   // DB193
{ S7_Optimized_Access := 'FALSE' }
// stored: AutoNumber false
   VAR
      L1 : String[80] := '                  M/s. LABORATE PHARMACEUTICALS INDIA LIMITED             ';
      L2 : String[80] := '               111, YAMUNA NAGAR ROAD, SATIWALA, PAONTA SAHIB,         ';
      L3 : String[80] := '               DISS.- SIRMOUR, HIMACHAL PRADESH - 173025 INDIA';
      L4 : String[80] := '              STERILIZING DEPYROGENATION TUNNEL (MODEL NO- SDT-C-5H)    ';
      L5 : String[80] := '              ----------------------------------------------------------';
      L6 : String[80] := '  EQUIPMENT ID        :';
      L7 : String[80] := '  PRODUCT NAME        :';
      L8 : String[80] := '  BATCH NO            :';
      L9 : String[80] := '                                                             DATE:  /  /       ';
      L10 : String[80] := '  PROCESS STARTED AT  :   :  :     ';
      L11 : String[80] := '  OPERATOR NAME       :';
      L12 : String[80] := '  TUNNEL MODE         :';
      L13 : String[80] := '  RECEIPE TYPE        :';
      L14 : String[80] := '-------------------------------------------------------------------------';
      L15 : String[80] := '  CONTROL TEMP (DEG.C)    :                   CONVEYOR SPEED (mm/min)   :     ';
      L16 : String[80] := '  CONVEYOR ON TEMP (DEG.C):                   CONVEYOR OFF TEMP (DEG.C) :    ';
      L17 : String[80] := '  SHUTDOWN TEMP (DEG.C)   :                   PRINTING INTERVAL (SEC)   :       ';
      L18 : String[80] := '                                            ';
      L19 : String[80] := '  CHECKED BY:                                 VERIFIED BY:';
      L20 : String[80] := '********************************************************************************';
      L21 : String[80] := '  DZ=DRYING ZONE            MHZ=MAIN HEATING ZONE   ST IN=STERILIZATION IN';
      L22 : String[80] := '  ST OUT=STERILIZATION OUT  CZ UP=COOLING ZONE UP   CZ DOWN=COOLING ZONE DOWN ';
      L23 : String[80] := '********************************************************************************';
      L24 : String[80] := '             :  CH-1  :  CH-2  :  CH-3  :  CH-4  :  CH-5  :  CH-6  :  CONVEYOR  ';
      L25 : String[90] := '     TIME    :  DZ    :  MHZ   :  ST IN :  ST OUT:  CZ UP :  CZDOWN:  SPEED ';
      L26 : String[80] := '             :  DEG.C :  DEG.C :  DEG.C :  DEG.C :  DEG.C :  DEG.C :  mm/min ';
      L27 : String[80] := '--------------------------------------------------------------------------------';
      L28 : String[80] := '    :  :                                                                     ';
      L29 : String[80] := '                                                                     ';
      L30 : String[80];
      L31 : String[80] := '               RECEIPE TYPE :                                                   ';
      L32 : String[80] := '--------------------------------------------------------------------------------';
      ALM1 : String[80] := '    :  :       EMERGENCY PRESSED ';
      ALM2 : String[80] := '    :  :       TURBIN VFD TRIP ';
      ALM3 : String[80] := '    :  :       CONVEYOR SUPPLY FAIL ';
      ALM4 : String[80] := '    :  :       LAF SUPPLY FAIL ';
      ALM5 : String[80] := '    :  :       TURBIN SUPPLY FAIL';
      ALM6 : String[80] := '    :  :       VAPOR EXHAUST SUPPLY FAIL';
      ALM7 : String[80] := '    :  :       HEATER SUPPLY FAIL';
      ALM8 : String[80] := '    :  :       TEMPERATURE OVERSHOOT';
      ALM9 : String[80] := '    :  :       VAPOUR EXHAUST TRIP';
      ALM10 : String[80] := '    :  :       SINGLE PHASE FAIL ';
      ALM11 : String[80] := '    :  :       DRYING ZONE PRESSURE LOW/PLEASE CHECK SENSOR OR BLOWER ';
      ALM12 : String[80] := '    :  :       COOLING ZONE PRESSURE LOW/PLEASE CHECK SENSOR OR BLOWER ';
      ALM13 : String[80] := '    :  :       STERILIZING  PREESURE LOW/PLEASE CHECK SENSOR OR TURBINE ';
      ALM14 : String[80] := '    :  :       CONVEYOR VFD OVERLOAD ';
      ALM15 : String[80] := '    :  :       MAIN HEAT RTD SENSOR FAIL ';
      ALM16 : String[80] := '    :  :       STERILE IN RTD SENSOR FAIL ';
      ALM17 : String[80] := '    :  :       STERILE OUT RTD SENSOR FAIL ';
      ALM18 : String[80] := '    :  :       CONVEYOR VFD TRIP ';
      ALM19 : String[80] := '    :  :       SHUTDOWN CYCLE STARTED ';
      ALM20 : String[80] := '    :  :                     *****PROCESS COMPLETED*****';
      ALM21 : String[80] := '  CHECKED BY:                                 VERIFIED BY:';
      "BATCH SIZE" : String[80] := '  BATCH SIZE          :';
      "CONTAINER SIZE" : String[80] := '  CONTAINER SIZE      :';
      "BLANK LINE" : String[80] := '                                                                ';
      ADDRESS : String[80] := ' ';
   END_VAR
BEGIN
END_DATA_BLOCK

DATA_BLOCK "PV"   // DB194
{ S7_Optimized_Access := 'TRUE' }
// stored: MemoryReserve 100
   VAR
      "CHAMBER PRESS" : Real;
      "DRAIN TEMP" : Real;
      "JACKET TEMP" : Real;
      VACCUM : Real;
      "CHAMBER TEMP1" : Real;
      "CHAMBER TEMP2" : Real;
      "CHAMBER TEMP3" : Real;
      "CHAMBER TEMP4" : Real;
      "DOOR1 PRESS" : Real;
      "DOOR2 PRESS" : Real;
      "JACKET PRESS" : Real;
      "DOOR1 VACCUM" : Real;
      "DOOR2 VACCUM" : Real;
      "JACKET VACCUM" : Real;
   END_VAR
BEGIN
END_DATA_BLOCK

DATA_BLOCK "RETAIN"   // DB81
{ S7_Optimized_Access := 'FALSE' }
   VAR RETAIN
      "CHAMBER PRESS SCL MAX" : Real := 5.0;
      "CHAMBER PRESS SCL MIN" : Real := -1.0;
      "JACKET PRESS SCL MAX" : Real := 5.0;
      "JACKET PRESS SCL MIN" : Real := -1.0;
      "CHAMBER VCC SCL MAX" : Real := 5.0;
      "CHAMBER VCC SCL MIN" : Real := -1.0;
      "SET PWD TEMP" : Real := 0.0;
      "SET CHAMBER PRESS HIGH" : Real := 1.25;
      "SET STERILE TEMP1" : Real := 105.0;
      "SET DRY VCC" : Real := -0.5;
      "SET STERILE EXH PRESS" : Real := 0.05;
      "SET ATM PRESS" : Real := -0.05;
      "SET EXIT TEMP" : Real := 101.0;
      "SET CHAMBER PRESS LOW" : Real := 1.18;
      "SET WFI TEMP" : Real := 0.0;
      "SET CONTROL BAND" : Real := 0.2;
      "SET STERILE TEMP2" : Real := 110.0;
      "SET STERILE TEMP3" : Real := 115.0;
      "SET STERILE TEMP4" : Real := 121.4;
      "SET LEAK VCC" : Real := -0.7;
      "SET VCC PRESS" : Real := -0.05;
      "SET STD1 TEMP1" : Real := 100.0;
      "SET STD1 TEMP2" : Real := 110.0;
      "SET STD1 TEMP3" : Real := 119.0;
      "SET STD1 PRESS" : Real := 0.05;
      "SET BOW VCC" : Real := -0.6;
      "SET BOW HEATUP" : Real := 121.4;
      "SET BOW EXH PRESS" : Real := 0.05;
      "SET BOW ATS PRESS" : Real := 0.0;
      "SET BOW END PRESS" : Real := -0.05;
      "SET BOW UP PRESS" : Real := 0.5;
      "SET HPHV VCC" : Real := -0.6;
      "SET HPHV HEATUP" : Real := 121.4;
      "SET HPHV EXH PRESS" : Real := 0.5;
      "SET HPHV ATS PRESS" : Real := -0.5;
      "SET HPHV END PRESS" : Real := -0.05;
      "SET HPHV UP PRESS" : Real := 0.5;
      "SET HZ" : Real := 25.0;
      "DOOR1 VCC SCL MIN" : Real := -1.0;
      "DOOR1 VCC SCL MAX" : Real := 5.0;
      "DOOR2 VCC SCL MIN" : Real := -1.0;
      "DOOR2 VCC SCL MAX" : Real := 5.0;
      "DOOR1 PRESS SCL MIN" : Real := -1.0;
      "DOOR1 PRESS SCL MAX" : Real := 5.0;
      "DOOR2 PRESS SCL MIN" : Real := -1.0;
      "DOOR2 PRESS SCL MAX" : Real := 5.0;
      "SET JACKET PRESS HIGH" : Real := 1.25;
      "SET DOOR1 PRESS HIGH" : Real := 2.55;
      "SET DOOR2 PRESS HIGH" : Real := 2.55;
      "SET DOOR1 VCC" : Real := -0.7;
      "SET DOOR2 VCC" : Real := -0.7;
      "SET JACKET LOW PRESS" : Real := 1.1;
      "SET DOOR1 PRESS LOW" : Real := 2.35;
      "SET DOOR2 PRESS LOW" : Real := 2.35;
      "SET PWD INLET TIME" : Int := 7;
      "SET DTG DSG TIME" : Int := 60;
      "SET PWD CRC TIME" : Int := 10;
      "SET PWD DRAIN" : Int := 7;
      "SET PRINT INTERVAL" : Int := 60;
      "SET WFI INLET TIME" : Int := 7;
      "SET WFI DSG TIME" : Int := 60;
      "SET WFI CRC TIME" : Int := 10;
      "SET WFI DRAIN TIME" : Int := 10;
      "SET WFI COUNTS" : Int := 0;
      "SET STERILE TIME1" : Int := 5;
      "SET STERILE TIME2" : Int := 5;
      "SET STERILE TIME3" : Int := 5;
      "SET STERILE TIME4" : Int := 30;
      "SET VENT TIME" : Int := 0;
      "SET VCC HOLD TIME" : Int := 10;
      "SET STD1 HOLD1" : Int := 5;
      "SET STD1 HOLD2" : Int := 3;
      "SET STD1 HOLD3" : Int := 2;
      "SET BOW  VCC HOLD TIME" : Int := 0;
      "SET NO OF BOW" : Int := 4;
      "SET BOW HEAT HOLD TIME" : Int := 10;
      "SET BOW ATS HOLD" : Int := 0;
      "SET DRY TIME" : Int := 20;
      "SET HPHV VCC HOLD" : Int := 0;
      "SET NO OF HPHV" : Int := 3;
      "SET HPHV HEAT HOLD" : Int := 10;
      "SET HPHV ATS HOLD" : Int := 5;
      "SET NO OF PWD" : Int := 2;
      "SET OFF EXHAUST" : Int := 40;
      "SET ON EXHAUST" : Int := 2;
      "SET STD1 VCC" : Real := 0.0;
      "SET STD1 UP PRESS" : Real := 0.0;
      "SET STD1 VCC HOLD" : Int := 0;
      "SET NO OF STD1 PULSE" : Int := 0;
      "SET STD2 TEMP1" : Real := 100.0;
      "SET STD2 TEMP2" : Real := 110.0;
      "SET STD2 TEMP3" : Real := 119.0;
      "SET STD2 PRESS" : Real := 0.05;
      "SET STD2 HOLD1" : Int := 5;
      "SET STD2 HOLD2" : Int := 3;
      "SET STD2 HOLD3" : Int := 2;
      "SET STD2 VCC" : Real := 0.0;
      "SET STD2 UP PRESS" : Real := 0.0;
      "SET STD2 VCC HOLD" : Int := 0;
      "SET NO OF STD2 PULSE" : Int := 0;
      "SET ACCEPTANCE LEAK" : Real := 0.013;
      "JACKET VCC SCL MIN" : Real := -1.0;
      "JACKET VCC SCL MAX" : Real := 5.0;
      "SET DELAY BEFORE HOLD" : Int := 3;
      "SET OVERSHOOT" : Real := 124.0;
      "SET ABORT TEMP" : Real := 120.5;
      DUMMY2 : Real := 0.0;
      DUMMY3 : Real := 0.0;
      DUMMY4 : Real := 0.0;
      DUMMY5 : Real := 0.0;
      DUMMY6 : Real := 0.0;
      "SET ABORT DELAY" : Int := 0;
      "SET WFI NO OF CYCLE" : Int := 0;
      "INT ATG3" : Int := 0;
      "INT ATG4" : Int := 0;
      "INT ATG5" : Int := 0;
      "INT ATG6" : Int := 0;
      "INT ATG7" : Int := 0;
      "INT ATG8" : Int := 0;
      "INT ATG9" : Int := 0;
      STD3 { S7_SetPoint := 'True'} : "STD";
      STD4 { S7_SetPoint := 'True'} : "STD";
      STD5 { S7_SetPoint := 'True'} : "STD";
      STD6 { S7_SetPoint := 'True'} : "STD";
      STD7 { S7_SetPoint := 'True'} : "STD";
      STD8 { S7_SetPoint := 'True'} : "STD";
      STD9 { S7_SetPoint := 'True'} : "STD";
      "SET BOILER ON TEMP" : Real := 133.0;
      "SET BOILER OFF TEMP" : Real := 135.0;
      "SET JACKET ON TIME" : Int := 10;
      "SET JACKET OFF TIME" : Int := 10;
      "SET BOILER WATER OFF DELAY" : Int := 25;
      "SET PRESSURE VERY HIGH" : Real := 1.3;
      "SET VACUUM BREAK FAIL TIME" : Int := 10;
      "SET JACKET PRESSURE HH" : Real := 1.4;
      "SET DOOR1 ALM PRESSURE" : Real := 0.3;
      "SET DOOR2 ALM PRESSURE" : Real := 0.3;
   END_VAR
BEGIN
   STD3."SET TEMP1" := 0.0;
   STD3."SET TEMP2" := 0.0;
   STD3."SET TEMP3" := 0.0;
   STD3."SET PRESS" := 0.0;
   STD3."SET HOLD1" := 0;
   STD3."SET HOLD2" := 0;
   STD3."SET HOLD3" := 0;
   STD3."SET VCC" := 0.0;
   STD3."SET UP PRESS" := 0.0;
   STD3."SET VCC HOLD" := 0;
   STD3."SET NO OF PULSE" := 0;
   STD4."SET TEMP1" := 0.0;
   STD4."SET TEMP2" := 0.0;
   STD4."SET TEMP3" := 0.0;
   STD4."SET PRESS" := 0.0;
   STD4."SET HOLD1" := 0;
   STD4."SET HOLD2" := 0;
   STD4."SET HOLD3" := 0;
   STD4."SET VCC" := 0.0;
   STD4."SET UP PRESS" := 0.0;
   STD4."SET VCC HOLD" := 0;
   STD4."SET NO OF PULSE" := 0;
   STD5."SET TEMP1" := 0.0;
   STD5."SET TEMP2" := 0.0;
   STD5."SET TEMP3" := 0.0;
   STD5."SET PRESS" := 0.0;
   STD5."SET HOLD1" := 0;
   STD5."SET HOLD2" := 0;
   STD5."SET HOLD3" := 0;
   STD5."SET VCC" := 0.0;
   STD5."SET UP PRESS" := 0.0;
   STD5."SET VCC HOLD" := 0;
   STD5."SET NO OF PULSE" := 0;
   STD6."SET TEMP1" := 0.0;
   STD6."SET TEMP2" := 0.0;
   STD6."SET TEMP3" := 0.0;
   STD6."SET PRESS" := 0.0;
   STD6."SET HOLD1" := 0;
   STD6."SET HOLD2" := 0;
   STD6."SET HOLD3" := 0;
   STD6."SET VCC" := 0.0;
   STD6."SET UP PRESS" := 0.0;
   STD6."SET VCC HOLD" := 0;
   STD6."SET NO OF PULSE" := 0;
   STD7."SET TEMP1" := 0.0;
   STD7."SET TEMP2" := 0.0;
   STD7."SET TEMP3" := 0.0;
   STD7."SET PRESS" := 0.0;
   STD7."SET HOLD1" := 0;
   STD7."SET HOLD2" := 0;
   STD7."SET HOLD3" := 0;
   STD7."SET VCC" := 0.0;
   STD7."SET UP PRESS" := 0.0;
   STD7."SET VCC HOLD" := 0;
   STD7."SET NO OF PULSE" := 0;
   STD8."SET TEMP1" := 0.0;
   STD8."SET TEMP2" := 0.0;
   STD8."SET TEMP3" := 0.0;
   STD8."SET PRESS" := 0.0;
   STD8."SET HOLD1" := 0;
   STD8."SET HOLD2" := 0;
   STD8."SET HOLD3" := 0;
   STD8."SET VCC" := 0.0;
   STD8."SET UP PRESS" := 0.0;
   STD8."SET VCC HOLD" := 0;
   STD8."SET NO OF PULSE" := 0;
   STD9."SET TEMP1" := 0.0;
   STD9."SET TEMP2" := 0.0;
   STD9."SET TEMP3" := 0.0;
   STD9."SET PRESS" := 0.0;
   STD9."SET HOLD1" := 0;
   STD9."SET HOLD2" := 0;
   STD9."SET HOLD3" := 0;
   STD9."SET VCC" := 0.0;
   STD9."SET UP PRESS" := 0.0;
   STD9."SET VCC HOLD" := 0;
   STD9."SET NO OF PULSE" := 0;
END_DATA_BLOCK

DATA_BLOCK "REVAMP"   // DB1
{ S7_Optimized_Access := 'FALSE' }
   VAR
      L1 : String[80] := '$L$R                       CLIENT:- M/s. KWALITY PHARMACEUTICALS LTD             ';
      L2 : String[80] := '$L$R 6TH MILE STONE, VILL.NAG KALAN, MAJITHA ROAD, AMRITSAR, PUNJAB-143601';
      L3 : String[80] := '$L$R                                    BATCH DATA';
      L4 : String[80] := '$L$R                                STEAM STERILIZER   ';
      L5 : String[80] := '$L$R             -----------------------------------------------------';
      L6 : String[80] := '$L$REQUIPMENT ID        :';
      L7 : String[80] := '$L$RPRODUCT NAME        :';
      L8 : String[80] := '$L$RBATCH NO            :';
      L9 : String[80] := '                                                             DATE: 04/05/2025';
      L10 : String[80] := '  PROCESS STARTED AT  :13:09:19';
      L11 : String[80] := '$L$ROPERATOR NAME       :';
      L12 : String[80] := '$L$RPROCESS                    :    ';
      L13 : String[80] := '$L$R        :';
      L14 : String[80] := '-------------';
      L15 : String[80] := '$L$R   ';
      L16 : String[80] := '$L$R                           CYCLE COMPLETED   ';
      L17 : String[80] := '$L$R                 ';
      L18 : String[80] := '$L$R                                          ';
      L19 : String[80] := '$L$R DONE BY  :                                 CHECKED BY :';
      L20 : String[80] := '$L$R******************************************************************************';
      L21 : String[80] := '$L$R DATE  :                                     DATE :';
      L22 : String[80] := '$L$R  SUMMARY OF VACUUM LEAK TEST  ';
      L23 : String[80] := '$L$R******************************************************************************';
      L24 : String[80] := '$L$R  TIME  : PRESSURE:  CH-1  :  CH-2  :  CH-3  :  CH-4  :  CH-5  :  STATUS      ';
      L25 : String[90] := '$L$R           :  DZ    :  MHZ   :  ST IN :  ST OUT:  CZ UP :  CZDOWN:  SPEED ';
      L26 : String[80] := '$L$R        :  BAR    :  DEG.C :  DEG.C :  DEG.C :  DEG.C :  DEG.C :   ';
      L27 : String[80] := '$L$R------------------------------------------------------------------------------';
      L28 : String[80] := '  13:09:20    1.032    116.2    120.6    119.9    119.4    120.2 HEATUP-1 HOLD';
      L29 : String[80] := '$L$R                                                                   ';
      L30 : String[80] := '$L$R------------------------------------------------------------------------------';
      L31 : String[80] := '               RECEIPE TYPE :                                                   ';
      L32 : String[80] := '--------------------------------------------------------------------------------';
      ALM1 : String[80] := '$L$R13  9 20';
      ALM2 : String[80] := '$L$R13  9 20';
      ALM3 : String[80] := '$L$R13  9 20';
      ALM4 : String[80] := '$L$R13  9 20';
      ALM5 : String[80] := '$L$R13  9 20';
      ALM6 : String[80] := '$L$R13  9 20';
      ALM7 : String[80] := '$L$R13  9 20';
      ALM8 : String[80] := '$L$R13  9 20';
      ALM9 : String[80] := '$L$R13  9 20';
      ALM10 : String[80] := '$L$R13  9 20';
      ALM11 : String[80] := '$L$R13  9 20';
      ALM12 : String[80] := '$L$R13  9 20';
      ALM13 : String[80] := '$L$R13  9 20';
      ALM14 : String[80] := '$L$R13  9 20';
      ALM15 : String[80] := '$L$R13  9 20';
      ALM16 : String[80] := '$L$R13  9 20';
      ALM17 : String[80] := '$L$R13  9 20';
      ALM18 : String[80] := '$L$R13  9 20';
      ALM19 : String[80] := '$L$R13  9 20';
      ALM20 : String[80] := '$L$R13  9 20';
      ALM21 : String[80] := '$L$RCHECKED BY              :                   VERIFIED BY               :';
      "BATCH SIZE" : String[80] := '  CYCLE NO            :';
      "CONTAINER SIZE" : String[80] := '  CONTAINER SIZE      :';
      "BLANK LINE" : String[80] := '                                                                ';
      ALM22 : String[80] := '    :  :       STABILIZING ZONE PRESSURE LOW/PLEASE CHECK GAUGE OR BLOWER ';
      zero : String[80] := '0';
      pv : String[80] := '';
      COLAN : String[80] := ':';
      T1 : String[80] := '13:';
      T2 : String[80] := '13:09';
      T3 : String[80] := '13:09:';
      T4 : String[80] := '13:09:20';
      T5 : String[80] := '';
      HOURS_P : String[80] := '13';
      MIN_P : String[80] := ' 9';
      SEC_P : String[80] := '20';
      HOURS_P_1 : String[80] := '13';
      MIN_P_1 : String[80] := '09';
      SEC_P_1 : String[80] := '20';
      CH1 : String[80] := ' 1.032';
      CH2 : String[80] := '116.2';
      CH3 : String[80] := '120.6';
      CH4 : String[80] := '119.9';
      CH5 : String[80] := '119.4';
      CH6 : String[80] := '120.2';
      CONVEYOR : String[80] := 'HEATUP-1 HOLD';
      SPACE_1 : String[80] := ' ';
      SPACE_2 : String[80] := '  ';
      SPACE_3 : String[80] := '   ';
      SPACE_4 : String[80] := '    ';
      C1 : String[80] := '  13:09:20    1.032    116.2    120.6    119.9    119.4    120.2 ';
      C2 : String[80] := '';
      C3 : String[80] := '';
      L10_2 : String[80] := '  PROCESS STARTED AT  :';
      L9_2 : String[80] := '                                                             DATE: ';
      DATE_P : String[80] := ' 4';
      MONTH_P : String[80] := ' 5';
      YEAR_P : String[80] := '2025';
      DATE_P_1 : String[80] := '04';
      MONTH_P_1 : String[80] := '05';
      YEAR_P_1 : String[80] := '2025';
      SLASH : String[80] := '/';
      "DATE CONCATE" : String[80] := '04/05/2025';
      ALM_P_1 : String[80] := '    EMERGENCY PRESSED ';
      ALM_P_2 : String[80] := '    TURBINE VFD TRIP ';
      ALM_P_3 : String[80] := '    CONVEYOR SUPPLY FAIL ';
      ALM_P_4 : String[80] := '     LAF SUPLY FAIL ';
      ALM_P_5 : String[80] := '    TURBINE SUPLY FAIL';
      ALM_P_6 : String[80] := '    VAPOR EXHAUST SUPLY FAIL';
      ALM_P_7 : String[80] := '    HEATER SUPLY FAIL';
      ALM_P_8 : String[80] := '    TEMPERATURE OVERSHOOT';
      ALM_P_9 : String[80] := '    VAPOUR EXHAUST TRIP';
      ALM_P_10 : String[80] := '    PHASE FAIL ';
      ALM_P_11 : String[80] := '    DRYING ZONE PRESSURE LOW/PLEASE CHECK GAUGE OR BLOWER ';
      ALM_P_12 : String[80] := '    COOLING ZONE PRESSURE LOW/PLEASE CHECK GAUGE OR BLOWER ';
      ALM_P_13 : String[80] := '    STERILIZING ZONE PREESURE LOW/PLEASE CHECK GAUGE OR TURBINE ';
      ALM_P_14 : String[80] := '    CONVEYOR VFD OVERLOAD ';
      ALM_P_15 : String[80] := '    MAIN HEAT RTD SENSOR FAIL ';
      ALM_P_16 : String[80] := '    STERILE IN RTD SENSOR FAIL ';
      ALM_P_17 : String[80] := '    STERILE OUT RTD SENSOR FAIL ';
      ALM_P_18 : String[80] := '    DROP IN STERLIZATION ZONE TEMPERATURE ';
      ALM_P_19 : String[80] := '    SHUTDOWN CYCLE STARTED ';
      ALM_P_20 : String[80] := '    *****PROCESS COMPLETED*****';
      ALM_P_22 : String[80] := '    STABILIZING ZONE PRESSURE LOW/PLEASE CHECK GAUGE OR BLOWER ';
      ADD2 : String[80] := '$L$R                  AMRITSAR-143001. P';
      "CYCLE STOP" : String[80] := '   ******CYCLE ABORTED****** ';
   END_VAR
BEGIN
END_DATA_BLOCK

DATA_BLOCK "SET VALUE"   // DB85
{ S7_Optimized_Access := 'FALSE' }
   VAR
      "PWD DOSING TIME" : String[80] := '  DOSING TIME (SEC)          :      60      ';
      "PWD WTR INLET TIME" : String[80] := '  WATER INLET TIME (MIN)     :       7     ';
      "PWD CRC TIME" : String[80] := '  CIRCULATION TIME (MIN)     :      10   ';
      "PWD DRAIN TIME" : String[80] := '  DRAIN TIME (MIN)           :       7    ';
      "STERILE TEMP1" : String[80] := '  HEAT UP-1 (DEG.C)          :    105.0  ';
      "STERILE TEMP2" : String[80] := '  HEAT UP-2 (DEG.C)          :    110.0  ';
      "STERILE TEMP3" : String[80] := '  HEAT UP-3 (DEG.C)          :    115.0  ';
      "STERILE TEMP4" : String[80] := '  STERILE TEMP (DEG.C)       :    121.4 ';
      "STERILE HOLD1" : String[80] := '  PULSE                      :       5    ';
      "STERILE HOLD2" : String[80] := '  PULSE                      :       5    ';
      "STERILE HOLD3" : String[80] := '  PULSE                      :       5    ';
      "STERILE HOLD4" : String[80] := '  HOLD TIME (MIN)            :      30    ';
      "WFI DSG TIME" : String[80] := '  DOSING TIME (SEC)          :      60 ';
      "WFI WTR TIME" : String[80] := '  WATER INLET TIME (MIN)     :       7 ';
      "WFI CRC TIME" : String[80] := '  CIRCULATION TIME (MIN)     :      10  ';
      "WFI DRAIN TIME" : String[80] := '  DRAIN TIME (MIN)           :      10  ';
      "STERILE EXH PRESS" : String[80] := '  EXHAUST PRESSURE (BAR)     :     0.05';
      "DRY VCC" : String[80] := '  VACUUM (BAR)               :    -0.500';
      "DRY VCC TIME" : String[80] := '  HOLD TIME (MIN)            :            ';
      "DRY ATS PRESSURE" : String[80] := '  ATMOSPHERIC PRESSURE (BAR) :    -0.050';
      "DRY TIME" : String[80] := '  DRYING TIME(MIN)           :      20     ';
      "PWD TEMP" : String[80] := '  PWD TEMP (DEG.C)           :     0.0    ';
      "STD TEMP1" : String[80] := '  HEAT UP-1 TEMPERATURE (DEG.C)         :   114.0       ';
      "STD TEMP2" : String[80] := '  HEAT UP-2 TEMPERATURE (DEG.C)         :   116.0       ';
      "STD TEMP3" : String[80] := '  HEAT UP-3 TEMPERATURE (DEG.C)         :   119.0       ';
      "STD TIME1" : String[80] := '  HEAT UP-1 HOLD TIME (MIN)             :      5     ';
      "STD TIME2" : String[80] := '  HEAT UP-2 HOLD TIME (MIN)             :      3     ';
      "STD TIME3" : String[80] := '  HEAT UP-3 HOLD TIME (MIN)             :      2     ';
      LEAK : String[80] := '  VACUUM (BAR)               :    -0.700';
      "DELAY BEFORE HOLD" : String[80] := '  DELAY BEFORE HOLD (MIN)    :       5';
      ACCEPTANCE : String[80] := '  ACCEPTANCE LEAKAGE (BAR)   :     0.013';
      "VCC HOLD" : String[80] := '  HOLD TIME (MIN)            :     10     ';
      "VCC PRESS" : String[80] := '  VENT PRESSURE (BAR)        :    -0.08';
      "HPHV VCC" : String[80] := '  PRE-VACUUM LEVEL (BAR)                :   -0.700      ';
      "HPHV VCC HOLD" : String[80] := '  PRE-VACUUM HOLD TIME (MIN)            :      3        ';
      "HPHV HEATUP" : String[80] := '  STERILIZATION TEMPERATURE (DEG.C)     :   121.4        ';
      "HPHV HEATUP HOLD" : String[80] := '  STERILIZATION HOLD TIME (MIN)         :     30       ';
      "HPHV NO" : String[80] := '  PRE-PULSE NUMBER                      :      3        ';
      "HPHV ATS" : String[80] := '  POST-VACUUM LEVEL (BAR)               :   -0.700      ';
      "HPHV ATS HOLD" : String[80] := '  POST-VACUUM HOLD TIME (MIN)           :     15        ';
      "HPHV EXH PRESS" : String[80] := '  EXHAUST PRESSURE (BAR)                :    0.2         ';
      "HPHV HEATUP PRESS" : String[80] := '  PRE-HEAT PRESSURE (BAR)               :    0.7        ';
      "HPHV END PRESS" : String[80] := '  END PRESSURE (BAR)                    :   -0.08       ';
      "BOW VCC" : String[80] := '  PRE-VACUUM LEVEL (BAR)                :   -0.700      ';
      "BOW VCC HOLD" : String[80] := '  PRE-VACUUM HOLD TIME (MIN)            :      3        ';
      "BOW HEATUP" : String[80] := '  STERILIZATION TEMPERATURE (DEG.C)     :   121.4        ';
      "BOW HEATUP HOLD" : String[80] := '  STERILIZATION HOLD TIME (MIN)         :     10       ';
      "BOW PRE PULSES" : String[80] := '  PRE-PULSE NUMBER                      :      3        ';
      "BOW POST VACUUM" : String[80] := '  POST-VACUUM LEVEL (BAR)               :    0.0        ';
      "BOW POST VACUUM HOLD" : String[80] := '  POST-VACUUM HOLD TIME (MIN)           :      0        ';   // 40:
      "BOW EXH PRESS" : String[80] := '  EXHAUST PRESSURE (BAR)                :    0.90        ';
      "BOW HEATUP PRESS" : String[80] := '  PRE-HEAT PRESSURE (BAR)               :    0.7        ';
      "BOW END PRESS" : String[80] := '  END PRESSURE (BAR)                    :    0.00       ';
      "STD UP PRESS" : String[80] := '  PRE PRESSURE (BAR)         :               0.00';
      "STD STOP TEMP" : String[80] := '  STERILIZATION STOP TEMP (DEG.C)       :   120.9     ';
      "STD VCC HOLD" : String[80] := '  VACUUM HOLD TIME (MIN)     :             ';
      "STD NO OF PULSES" : String[80] := '  NO OF PULSES               :                 0';
      "DONE BY" : String[80] := '';
      "DATE" : String[80] := '';
      SUMARY : String[80] := '';
      "VACUUM START" : String[80] := '';
      "VACCUM END" : String[80] := '';
      "ACTUAL LEAK" : String[80] := '';
      "ACCEPT LEAK" : String[80] := '';
      RESULT : String[80] := '';
      "PW NO OF PULSES_1" : String[80] := '$L$RNO OF PULSES               :       2         ';
      "OVERSHOOT TEMP" : String[80] := '$L$ROVERSHOOT TEMP (DEG.C)                :   124.0      ';
      "ABORT TEMP" : String[80] := '$L$RCRITICAL TEMP (DEG.C)                 :   120.5          ';
      "ABORT DELAY" : String[80] := '$L$RABORT DELAY (SEC)          :       1       ';
      "SET WFI COUNTS" : String[80] := '$L$RNO OF PULSES               :       0        ';
      "SET HPHV HT1" : String[80] := '  HEAT UP-1 TEMPEARUTRE (DEG.C)         :   114.0       ';
      "SET HPHV HT2" : String[80] := '  HEAT UP-2 TEMPEARUTRE (DEG.C)         :   116.0       ';
      "SET HPHV HT3" : String[80] := '  HEAT UP-3 TEMPEARUTRE (DEG.C)         :   119.0        ';
      "SET HPHV UP T1" : String[80] := '  HEAT UP-1 HOLD TIME (MIN)             :      5     ';
      "SET HPHV UP T2" : String[80] := '  HEAT UP-2 HOLD TIME (MIN)             :      3     ';
      "SET HPHV UP T3" : String[80] := '  HEAT UP-3 HOLD TIME (MIN)             :      2     ';
      "SET BOW HT1" : String[80] := '  HEAT UP-1 TEMPEARUTRE (DEG.C)         :   114.0     ';
      "SET BOW HT2" : String[80] := '  HEAT UP-2 TEMPEARUTRE (DEG.C)         :   116.0      ';
      "SET BOW HT3" : String[80] := '  HEAT UP-3 TEMPEARUTRE (DEG.C)         :   119.0      ';
      "SET BOW UP T1" : String[80] := '  HEAT UP-1 HOLD TIME (MIN)             :      5     ';
      "SET BOW UP T2" : String[80] := '  HEAT UP-2 HOLD TIME (MIN)             :      3     ';
      "SET BOW UP T3" : String[80] := '  HEAT UP-3 HOLD TIME (MIN)             :      2     ';
      "SET HPHV POST PULSES" : String[80] := '  POST-PULSE NUMBER                     :      1        ';
      "SET BOW POST PULSES" : String[80] := '  POST-PULSE NUMBER                     :      0        ';
      "SET BOW STOP TMP" : String[80] := '  STERILIZATION STOP TEMP (DEG.C)       :   120.9     ';   // :41
      "SET HPHV STOP TMP" : String[80] := '  STERILIZATION STOP TEMP (DEG.C)       :   120.9     ';
      "CONTROL BAND" : String[80] := '  CONTROL BAND TEMP (DEG.C)             :     0.2         ';
      "JACKET ALM TIME" : String[80] := '  JACKET ALARM TIME (MIN)               :     10                   ';
      "HEAT ALM TIME" : String[80] := '  HEATUP ALARM TIME (MIN)               :     10                   ';
      "PRINT INTERVAL" : String[80] := '  PRINT INTERVAL TIME (SEC)             :     60               ';
      "STD STERILE TEMP" : String[80] := '  STERILIZATION TEMPERATURE (DEG.C)     :   121.4        ';
      "STD STERILE HOLD" : String[80] := '  STERILIZATION HOLD TIME (MIN)         :     10       ';
      "STD END PRESSURE" : String[80] := '  END PRESSURE (BAR)                    :    0.08       ';
      AMP_LEAK : String[80] := '  VACUUM (BAR)               :    -0.700';
      "AMPVCC HOLD" : String[80] := '  HOLD TIME (MIN)            :     10     ';
      "AMP VCC PRESS" : String[80] := '  VENT PRESSURE (BAR)        :    -0.08';
   END_VAR
BEGIN
END_DATA_BLOCK

DATA_BLOCK "new"   // DB260
{ S7_Optimized_Access := 'FALSE' }
   VAR RETAIN
      "std end press" : String[80] := '$L$REND PRESSURE (BAR)                    :               ';
      "STD STERILE HOLD TEMP" : Array[0..12] of Real;
      "STD STERILE HOLD TIME" : Array[0..12] of Int;
      "STD BAND" : Array[0..12] of Real;
      "STD OVER TEMP" : Array[0..12] of Real;
      "STD ABORT TEMP" : Array[0..12] of Real;
      "STD STERILE STOP TEMP" : Array[0..12] of Real;
      "EXTRA TEMP" : Real := 0.3;
      "HPHV SET TEMP" : Array[0..3] of Real;
      "BOW SET TEMP" : Array[0..3] of Real;
      "HPHV SET TIME" : Array[0..3] of Int;
      "BOW SET TIME" : Array[0..3] of Int;
      "HPHV STOP TEMP" : Real := 120.9;
      "BOW STOP TEMP" : Real := 120.9;
      "JACKET ALARM TIME" : Int := 10;
      "HEATUP ALARM TIME" : Int := 10;
      "TEMP OFFSET" : Array[0..10] of Real;
      "SET VACUUM ALARM TIME" : Int := 30;
      "SET LEAK VCC" : Real := -0.7;
      "SET VCC PRESS" : Real := -0.05;
      "SET DELAY BEFORE HOLD TIME" : Int := 0;
      "SET VCC HOLD TIME" : Int := 10;
      "SET ACCEPTANCE LEAK" : Real := 0.013;
   END_VAR
BEGIN
   "STD STERILE HOLD TEMP"[0..2] := 121.4;
   "STD STERILE HOLD TEMP"[3..5] := 115.0;
   "STD STERILE HOLD TEMP"[6] := 110.0;
   "STD STERILE HOLD TEMP"[7..8] := 100.0;
   "STD STERILE HOLD TEMP"[9..12] := 0.0;
   "STD STERILE HOLD TIME"[0] := 30;
   "STD STERILE HOLD TIME"[1] := 20;
   "STD STERILE HOLD TIME"[2] := 15;
   "STD STERILE HOLD TIME"[3] := 35;
   "STD STERILE HOLD TIME"[4] := 30;
   "STD STERILE HOLD TIME"[5..6] := 15;
   "STD STERILE HOLD TIME"[7] := 35;
   "STD STERILE HOLD TIME"[8] := 20;
   "STD STERILE HOLD TIME"[9..12] := 0;
   "STD BAND"[0..12] := 0.0;
   "STD OVER TEMP"[0..2] := 124.0;
   "STD OVER TEMP"[3..5] := 118.0;
   "STD OVER TEMP"[6] := 113.0;
   "STD OVER TEMP"[7..8] := 103.0;
   "STD OVER TEMP"[9..10] := 124.0;
   "STD OVER TEMP"[11..12] := 0.0;
   "STD ABORT TEMP"[0..2] := 120.5;
   "STD ABORT TEMP"[3..5] := 114.5;
   "STD ABORT TEMP"[6..7] := 109.5;
   "STD ABORT TEMP"[8] := 99.5;
   "STD ABORT TEMP"[9..10] := 120.5;
   "STD ABORT TEMP"[11..12] := 0.0;
   "STD STERILE STOP TEMP"[0..2] := 120.9;
   "STD STERILE STOP TEMP"[3..5] := 114.9;
   "STD STERILE STOP TEMP"[6] := 109.9;
   "STD STERILE STOP TEMP"[7..8] := 99.9;
   "STD STERILE STOP TEMP"[9..12] := 0.0;
   "HPHV SET TEMP"[0] := 114.0;
   "HPHV SET TEMP"[1] := 116.0;
   "HPHV SET TEMP"[2] := 119.0;
   "HPHV SET TEMP"[3] := 0.0;
   "BOW SET TEMP"[0] := 114.0;
   "BOW SET TEMP"[1] := 116.0;
   "BOW SET TEMP"[2] := 119.0;
   "BOW SET TEMP"[3] := 0.0;
   "HPHV SET TIME"[0] := 5;
   "HPHV SET TIME"[1] := 3;
   "HPHV SET TIME"[2] := 2;
   "HPHV SET TIME"[3] := 1;
   "BOW SET TIME"[0] := 5;
   "BOW SET TIME"[1] := 3;
   "BOW SET TIME"[2] := 2;
   "BOW SET TIME"[3] := 0;
   "TEMP OFFSET"[0..1] := 0.0;
   "TEMP OFFSET"[2..3] := 0.2;
   "TEMP OFFSET"[4] := 0.0;
   "TEMP OFFSET"[5] := 0.1;
   "TEMP OFFSET"[6..10] := 0.0;
END_DATA_BLOCK

ORGANIZATION_BLOCK "Main"   // OB1, LAD, ProgramCycle
TITLE = "Main Program Sweep (Cycle)"
{ S7_Optimized_Access := 'TRUE' }
// stored: SetENOAutomatically false
   VAR_INPUT
      Initial_Call : Bool;   // Initial call of this OB
      Remanence : Bool;   // =True, if remanent data are available
   END_VAR
   VAR_TEMP
      "EQUIPMENT ID" : Variant;
      "EQUIPMENT ID_1" : Variant;
   END_VAR
   VAR_TEMP   // added for the SCL form of the ladder/FBD networks
      _w1 : Bool;
      _w2 : Bool;
      _w3 : Bool;
      _w4 : Bool;
      _w5 : Bool;
      _w6 : Bool;
      _w7 : Bool;
   END_VAR
BEGIN

REGION Network 1: BLOCK CALL
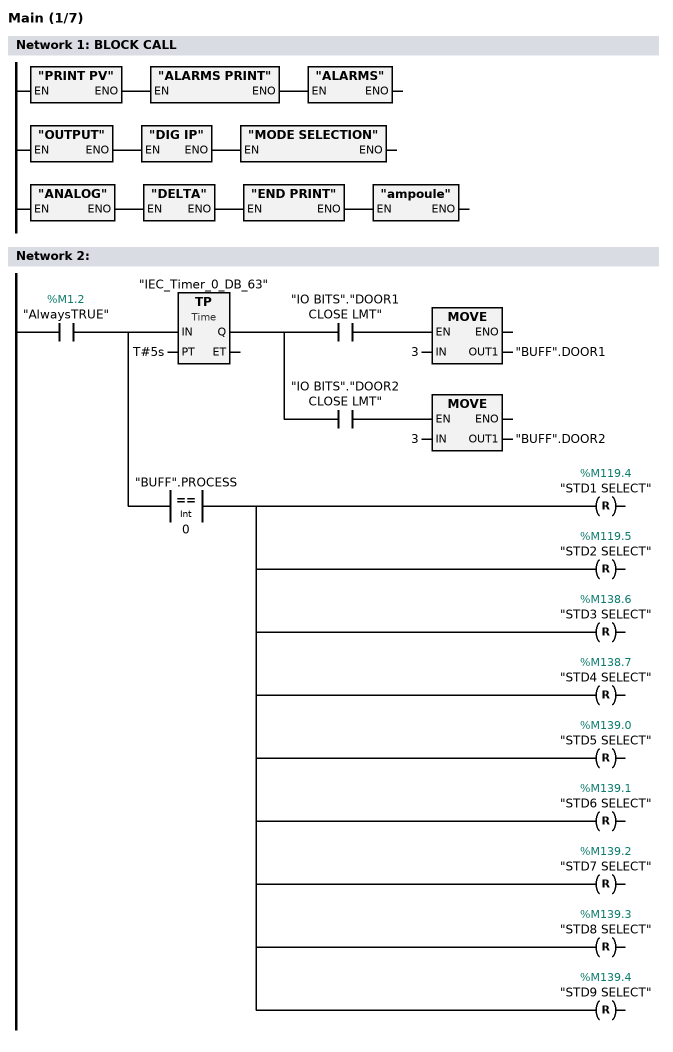
   RUNG wire#powerrail
      "PRINT PV"()
      "ALARMS PRINT"()
      "ALARMS"()
   END_RUNG
   RUNG wire#powerrail
      "OUTPUT"()
      "DIG IP"()
      "MODE SELECTION"()
   END_RUNG
   RUNG wire#powerrail
      "ANALOG"()
      "DELTA"()
      "END PRINT"()
      "ampoule"()
   END_RUNG
   // the same network as SCL:
   "PRINT PV"(ENO => #_w1);
   "ALARMS PRINT"(EN := #_w1, ENO => #_w2);
   IF #_w2 THEN "ALARMS"(); END_IF;
   "OUTPUT"(ENO => #_w3);
   "DIG IP"(EN := #_w3, ENO => #_w4);
   IF #_w4 THEN "MODE SELECTION"(); END_IF;
   "ANALOG"(ENO => #_w5);
   "DELTA"(EN := #_w5, ENO => #_w6);
   "END PRINT"(EN := #_w6, ENO => #_w7);
   IF #_w7 THEN "ampoule"(); END_IF;
END_REGION

REGION Network 2
   RUNG wire#powerrail
      Contact( "AlwaysTRUE" )
      wire#w1
      { S7_Templates := "time_type := Time" } "IEC_Timer_0_DB_63".TP(pt := T#5s, et =>)
      wire#w2
      Contact( "IO BITS"."DOOR1 CLOSE LMT" )
      Move(in := 3, out1 => "BUFF".DOOR1)
   END_RUNG
   RUNG wire#w2
      Contact( "IO BITS"."DOOR2 CLOSE LMT" )
      Move(in := 3, out1 => "BUFF".DOOR2)
   END_RUNG
   RUNG wire#w1
      { S7_Templates := "SrcType := Int" } EQ_Contact(in1 := "BUFF".PROCESS, in2 := 0)
      wire#w3
      R_Coil( "STD1 SELECT" )
   END_RUNG
   RUNG wire#w3
      R_Coil( "STD2 SELECT" )
   END_RUNG
   RUNG wire#w3
      R_Coil( "STD3 SELECT" )
   END_RUNG
   RUNG wire#w3
      R_Coil( "STD4 SELECT" )
   END_RUNG
   RUNG wire#w3
      R_Coil( "STD5 SELECT" )
   END_RUNG
   RUNG wire#w3
      R_Coil( "STD6 SELECT" )
   END_RUNG
   RUNG wire#w3
      R_Coil( "STD7 SELECT" )
   END_RUNG
   RUNG wire#w3
      R_Coil( "STD8 SELECT" )
   END_RUNG
   RUNG wire#w3
      R_Coil( "STD9 SELECT" )
   END_RUNG
   // the same network as SCL:
   "IEC_Timer_0_DB_63".TP(IN := "AlwaysTRUE", PT := T#5s);
   IF "IEC_Timer_0_DB_63".Q AND "IO BITS"."DOOR1 CLOSE LMT" THEN "BUFF".DOOR1 := 3; END_IF;
   IF "IEC_Timer_0_DB_63".Q AND "IO BITS"."DOOR2 CLOSE LMT" THEN "BUFF".DOOR2 := 3; END_IF;
   IF "AlwaysTRUE" AND ("BUFF".PROCESS = 0) THEN
       "STD1 SELECT" := FALSE;
       "STD2 SELECT" := FALSE;
       "STD3 SELECT" := FALSE;
       "STD4 SELECT" := FALSE;
       "STD5 SELECT" := FALSE;
       "STD6 SELECT" := FALSE;
       "STD7 SELECT" := FALSE;
       "STD8 SELECT" := FALSE;
       "STD9 SELECT" := FALSE;
   END_IF;
END_REGION

REGION Network 3: STANDARD1
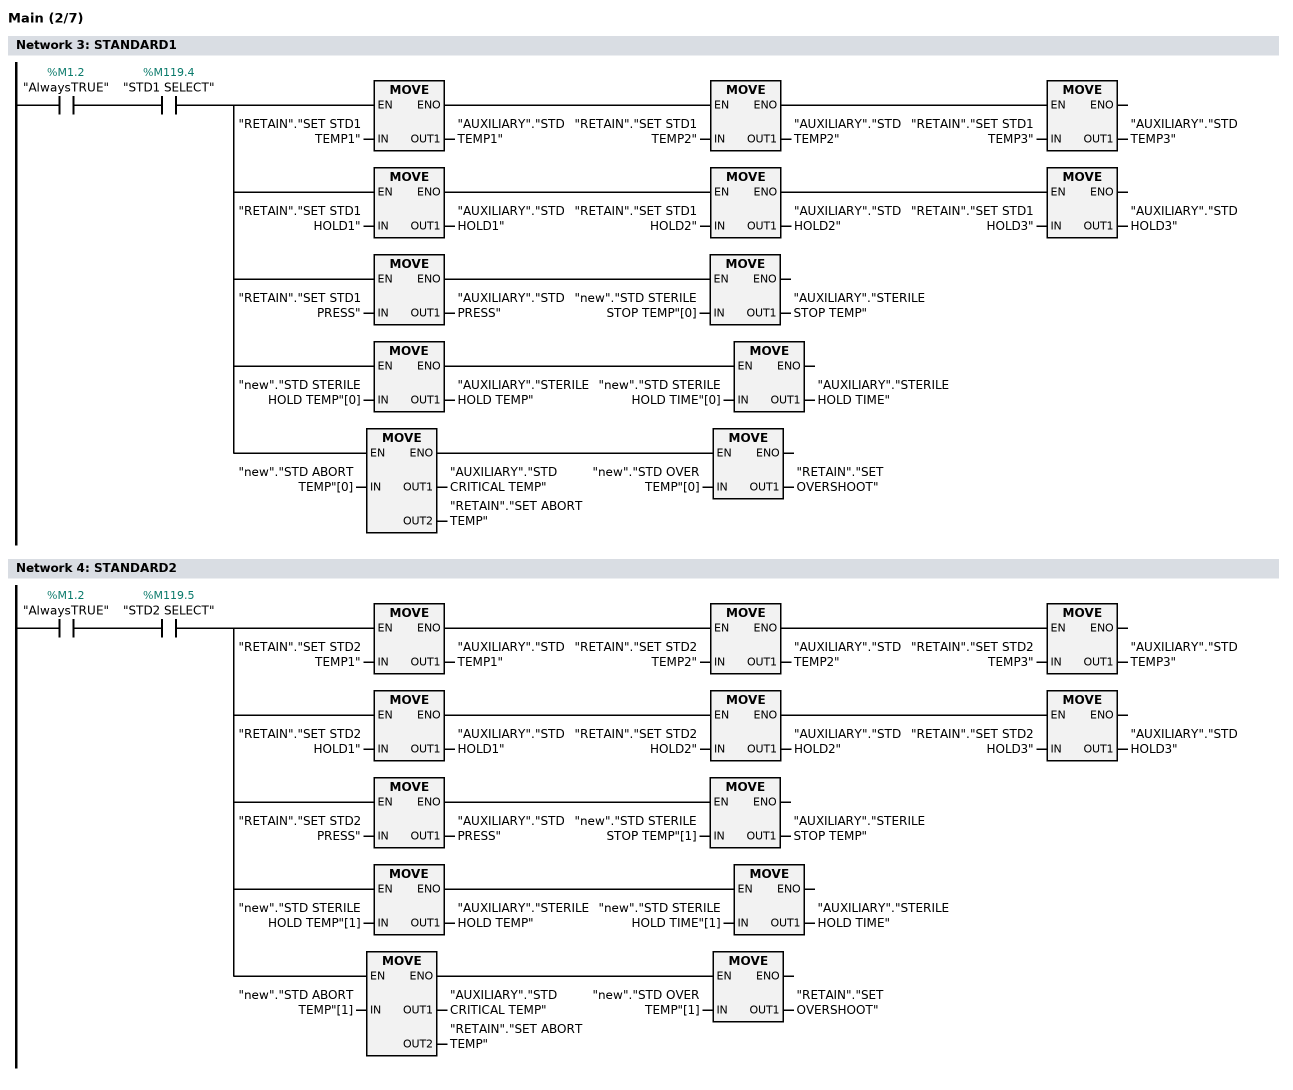
   RUNG wire#powerrail
      Contact( "AlwaysTRUE" )
      Contact( "STD1 SELECT" )
      wire#w1
      Move(in := "RETAIN"."SET STD1 TEMP1", out1 => "AUXILIARY"."STD TEMP1")
      Move(in := "RETAIN"."SET STD1 TEMP2", out1 => "AUXILIARY"."STD TEMP2")
      Move(in := "RETAIN"."SET STD1 TEMP3", out1 => "AUXILIARY"."STD TEMP3")
   END_RUNG
   RUNG wire#w1
      Move(in := "RETAIN"."SET STD1 HOLD1", out1 => "AUXILIARY"."STD HOLD1")
      Move(in := "RETAIN"."SET STD1 HOLD2", out1 => "AUXILIARY"."STD HOLD2")
      Move(in := "RETAIN"."SET STD1 HOLD3", out1 => "AUXILIARY"."STD HOLD3")
   END_RUNG
   RUNG wire#w1
      Move(in := "RETAIN"."SET STD1 PRESS", out1 => "AUXILIARY"."STD PRESS")
      Move(in := "new"."STD STERILE STOP TEMP"[0], out1 => "AUXILIARY"."STERILE STOP TEMP")
   END_RUNG
   RUNG wire#w1
      Move(in := "new"."STD STERILE HOLD TEMP"[0], out1 => "AUXILIARY"."STERILE HOLD TEMP")
      Move(in := "new"."STD STERILE HOLD TIME"[0], out1 => "AUXILIARY"."STERILE HOLD TIME")
   END_RUNG
   RUNG wire#w1
      Move(in := "new"."STD ABORT TEMP"[0], out1 => "AUXILIARY"."STD CRITICAL TEMP", out2 => "RETAIN"."SET ABORT TEMP")
      Move(in := "new"."STD OVER TEMP"[0], out1 => "RETAIN"."SET OVERSHOOT")
   END_RUNG
   // the same network as SCL:
   IF "AlwaysTRUE" AND "STD1 SELECT" THEN
       "AUXILIARY"."STD TEMP1" := "RETAIN"."SET STD1 TEMP1";
       "AUXILIARY"."STD TEMP2" := "RETAIN"."SET STD1 TEMP2";
       "AUXILIARY"."STD TEMP3" := "RETAIN"."SET STD1 TEMP3";
       "AUXILIARY"."STD HOLD1" := "RETAIN"."SET STD1 HOLD1";
       "AUXILIARY"."STD HOLD2" := "RETAIN"."SET STD1 HOLD2";
       "AUXILIARY"."STD HOLD3" := "RETAIN"."SET STD1 HOLD3";
       "AUXILIARY"."STD PRESS" := "RETAIN"."SET STD1 PRESS";
       "AUXILIARY"."STERILE STOP TEMP" := "new"."STD STERILE STOP TEMP"[0];
       "AUXILIARY"."STERILE HOLD TEMP" := "new"."STD STERILE HOLD TEMP"[0];
       "AUXILIARY"."STERILE HOLD TIME" := "new"."STD STERILE HOLD TIME"[0];
       "AUXILIARY"."STD CRITICAL TEMP" := "new"."STD ABORT TEMP"[0];
       "RETAIN"."SET ABORT TEMP" := "new"."STD ABORT TEMP"[0];
       "RETAIN"."SET OVERSHOOT" := "new"."STD OVER TEMP"[0];
   END_IF;
END_REGION

REGION Network 4: STANDARD2
   RUNG wire#powerrail
      Contact( "AlwaysTRUE" )
      Contact( "STD2 SELECT" )
      wire#w1
      Move(in := "RETAIN"."SET STD2 TEMP1", out1 => "AUXILIARY"."STD TEMP1")
      Move(in := "RETAIN"."SET STD2 TEMP2", out1 => "AUXILIARY"."STD TEMP2")
      Move(in := "RETAIN"."SET STD2 TEMP3", out1 => "AUXILIARY"."STD TEMP3")
   END_RUNG
   RUNG wire#w1
      Move(in := "RETAIN"."SET STD2 HOLD1", out1 => "AUXILIARY"."STD HOLD1")
      Move(in := "RETAIN"."SET STD2 HOLD2", out1 => "AUXILIARY"."STD HOLD2")
      Move(in := "RETAIN"."SET STD2 HOLD3", out1 => "AUXILIARY"."STD HOLD3")
   END_RUNG
   RUNG wire#w1
      Move(in := "RETAIN"."SET STD2 PRESS", out1 => "AUXILIARY"."STD PRESS")
      Move(in := "new"."STD STERILE STOP TEMP"[1], out1 => "AUXILIARY"."STERILE STOP TEMP")
   END_RUNG
   RUNG wire#w1
      Move(in := "new"."STD STERILE HOLD TEMP"[1], out1 => "AUXILIARY"."STERILE HOLD TEMP")
      Move(in := "new"."STD STERILE HOLD TIME"[1], out1 => "AUXILIARY"."STERILE HOLD TIME")
   END_RUNG
   RUNG wire#w1
      Move(in := "new"."STD ABORT TEMP"[1], out1 => "AUXILIARY"."STD CRITICAL TEMP", out2 => "RETAIN"."SET ABORT TEMP")
      Move(in := "new"."STD OVER TEMP"[1], out1 => "RETAIN"."SET OVERSHOOT")
   END_RUNG
   // the same network as SCL:
   IF "AlwaysTRUE" AND "STD2 SELECT" THEN
       "AUXILIARY"."STD TEMP1" := "RETAIN"."SET STD2 TEMP1";
       "AUXILIARY"."STD TEMP2" := "RETAIN"."SET STD2 TEMP2";
       "AUXILIARY"."STD TEMP3" := "RETAIN"."SET STD2 TEMP3";
       "AUXILIARY"."STD HOLD1" := "RETAIN"."SET STD2 HOLD1";
       "AUXILIARY"."STD HOLD2" := "RETAIN"."SET STD2 HOLD2";
       "AUXILIARY"."STD HOLD3" := "RETAIN"."SET STD2 HOLD3";
       "AUXILIARY"."STD PRESS" := "RETAIN"."SET STD2 PRESS";
       "AUXILIARY"."STERILE STOP TEMP" := "new"."STD STERILE STOP TEMP"[1];
       "AUXILIARY"."STERILE HOLD TEMP" := "new"."STD STERILE HOLD TEMP"[1];
       "AUXILIARY"."STERILE HOLD TIME" := "new"."STD STERILE HOLD TIME"[1];
       "AUXILIARY"."STD CRITICAL TEMP" := "new"."STD ABORT TEMP"[1];
       "RETAIN"."SET ABORT TEMP" := "new"."STD ABORT TEMP"[1];
       "RETAIN"."SET OVERSHOOT" := "new"."STD OVER TEMP"[1];
   END_IF;
END_REGION

REGION Network 5: STANDARD3
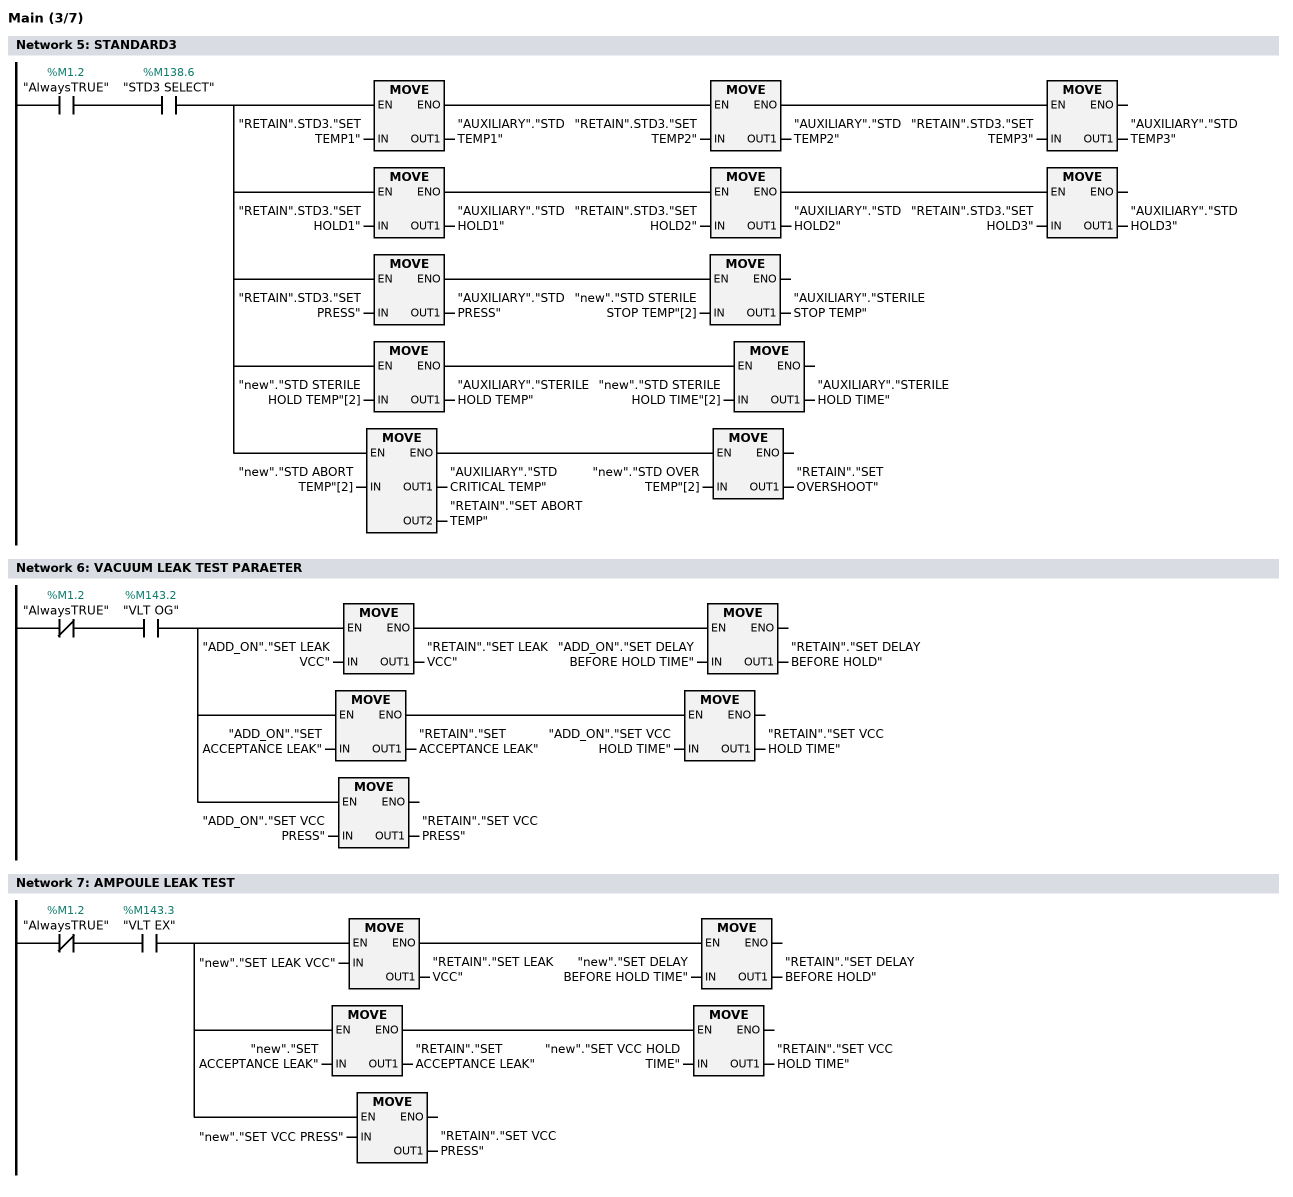
   RUNG wire#powerrail
      Contact( "AlwaysTRUE" )
      Contact( "STD3 SELECT" )
      wire#w1
      Move(in := "RETAIN".STD3."SET TEMP1", out1 => "AUXILIARY"."STD TEMP1")
      Move(in := "RETAIN".STD3."SET TEMP2", out1 => "AUXILIARY"."STD TEMP2")
      Move(in := "RETAIN".STD3."SET TEMP3", out1 => "AUXILIARY"."STD TEMP3")
   END_RUNG
   RUNG wire#w1
      Move(in := "RETAIN".STD3."SET HOLD1", out1 => "AUXILIARY"."STD HOLD1")
      Move(in := "RETAIN".STD3."SET HOLD2", out1 => "AUXILIARY"."STD HOLD2")
      Move(in := "RETAIN".STD3."SET HOLD3", out1 => "AUXILIARY"."STD HOLD3")
   END_RUNG
   RUNG wire#w1
      Move(in := "RETAIN".STD3."SET PRESS", out1 => "AUXILIARY"."STD PRESS")
      Move(in := "new"."STD STERILE STOP TEMP"[2], out1 => "AUXILIARY"."STERILE STOP TEMP")
   END_RUNG
   RUNG wire#w1
      Move(in := "new"."STD STERILE HOLD TEMP"[2], out1 => "AUXILIARY"."STERILE HOLD TEMP")
      Move(in := "new"."STD STERILE HOLD TIME"[2], out1 => "AUXILIARY"."STERILE HOLD TIME")
   END_RUNG
   RUNG wire#w1
      Move(in := "new"."STD ABORT TEMP"[2], out1 => "AUXILIARY"."STD CRITICAL TEMP", out2 => "RETAIN"."SET ABORT TEMP")
      Move(in := "new"."STD OVER TEMP"[2], out1 => "RETAIN"."SET OVERSHOOT")
   END_RUNG
   // the same network as SCL:
   IF "AlwaysTRUE" AND "STD3 SELECT" THEN
       "AUXILIARY"."STD TEMP1" := "RETAIN".STD3."SET TEMP1";
       "AUXILIARY"."STD TEMP2" := "RETAIN".STD3."SET TEMP2";
       "AUXILIARY"."STD TEMP3" := "RETAIN".STD3."SET TEMP3";
       "AUXILIARY"."STD HOLD1" := "RETAIN".STD3."SET HOLD1";
       "AUXILIARY"."STD HOLD2" := "RETAIN".STD3."SET HOLD2";
       "AUXILIARY"."STD HOLD3" := "RETAIN".STD3."SET HOLD3";
       "AUXILIARY"."STD PRESS" := "RETAIN".STD3."SET PRESS";
       "AUXILIARY"."STERILE STOP TEMP" := "new"."STD STERILE STOP TEMP"[2];
       "AUXILIARY"."STERILE HOLD TEMP" := "new"."STD STERILE HOLD TEMP"[2];
       "AUXILIARY"."STERILE HOLD TIME" := "new"."STD STERILE HOLD TIME"[2];
       "AUXILIARY"."STD CRITICAL TEMP" := "new"."STD ABORT TEMP"[2];
       "RETAIN"."SET ABORT TEMP" := "new"."STD ABORT TEMP"[2];
       "RETAIN"."SET OVERSHOOT" := "new"."STD OVER TEMP"[2];
   END_IF;
END_REGION

REGION Network 6: VACUUM LEAK TEST PARAETER
   RUNG wire#powerrail
      I_Contact( "AlwaysTRUE" )
      Contact( "VLT OG" )
      wire#w1
      Move(in := "ADD_ON"."SET LEAK VCC", out1 => "RETAIN"."SET LEAK VCC")
      Move(in := "ADD_ON"."SET DELAY BEFORE HOLD TIME", out1 => "RETAIN"."SET DELAY BEFORE HOLD")
   END_RUNG
   RUNG wire#w1
      Move(in := "ADD_ON"."SET ACCEPTANCE LEAK", out1 => "RETAIN"."SET ACCEPTANCE LEAK")
      Move(in := "ADD_ON"."SET VCC HOLD TIME", out1 => "RETAIN"."SET VCC HOLD TIME")
   END_RUNG
   RUNG wire#w1
      Move(in := "ADD_ON"."SET VCC PRESS", out1 => "RETAIN"."SET VCC PRESS")
   END_RUNG
   // the same network as SCL:
   IF NOT "AlwaysTRUE" AND "VLT OG" THEN
       "RETAIN"."SET LEAK VCC" := "ADD_ON"."SET LEAK VCC";
       "RETAIN"."SET DELAY BEFORE HOLD" := "ADD_ON"."SET DELAY BEFORE HOLD TIME";
       "RETAIN"."SET ACCEPTANCE LEAK" := "ADD_ON"."SET ACCEPTANCE LEAK";
       "RETAIN"."SET VCC HOLD TIME" := "ADD_ON"."SET VCC HOLD TIME";
       "RETAIN"."SET VCC PRESS" := "ADD_ON"."SET VCC PRESS";
   END_IF;
END_REGION

REGION Network 7: AMPOULE LEAK TEST
   RUNG wire#powerrail
      I_Contact( "AlwaysTRUE" )
      Contact( "VLT EX" )
      wire#w1
      Move(in := "new"."SET LEAK VCC", out1 => "RETAIN"."SET LEAK VCC")
      Move(in := "new"."SET DELAY BEFORE HOLD TIME", out1 => "RETAIN"."SET DELAY BEFORE HOLD")
   END_RUNG
   RUNG wire#w1
      Move(in := "new"."SET ACCEPTANCE LEAK", out1 => "RETAIN"."SET ACCEPTANCE LEAK")
      Move(in := "new"."SET VCC HOLD TIME", out1 => "RETAIN"."SET VCC HOLD TIME")
   END_RUNG
   RUNG wire#w1
      Move(in := "new"."SET VCC PRESS", out1 => "RETAIN"."SET VCC PRESS")
   END_RUNG
   // the same network as SCL:
   IF NOT "AlwaysTRUE" AND "VLT EX" THEN
       "RETAIN"."SET LEAK VCC" := "new"."SET LEAK VCC";
       "RETAIN"."SET DELAY BEFORE HOLD" := "new"."SET DELAY BEFORE HOLD TIME";
       "RETAIN"."SET ACCEPTANCE LEAK" := "new"."SET ACCEPTANCE LEAK";
       "RETAIN"."SET VCC HOLD TIME" := "new"."SET VCC HOLD TIME";
       "RETAIN"."SET VCC PRESS" := "new"."SET VCC PRESS";
   END_IF;
END_REGION

REGION Network 8: MONTH_L
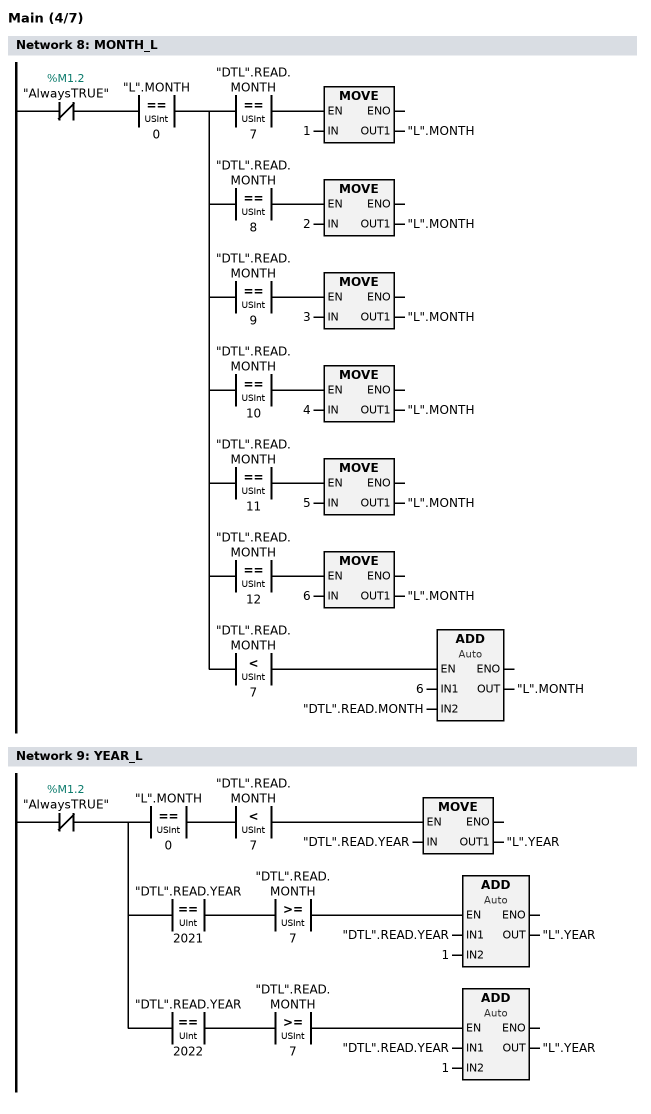
   RUNG wire#powerrail
      I_Contact( "AlwaysTRUE" )
      { S7_Templates := "SrcType := USInt" } EQ_Contact(in1 := "L".MONTH, in2 := 0)
      wire#w1
      { S7_Templates := "SrcType := USInt" } EQ_Contact(in1 := "DTL".READ.MONTH, in2 := 7)
      Move(in := 1, out1 => "L".MONTH)
   END_RUNG
   RUNG wire#w1
      { S7_Templates := "SrcType := USInt" } EQ_Contact(in1 := "DTL".READ.MONTH, in2 := 8)
      Move(in := 2, out1 => "L".MONTH)
   END_RUNG
   RUNG wire#w1
      { S7_Templates := "SrcType := USInt" } EQ_Contact(in1 := "DTL".READ.MONTH, in2 := 9)
      Move(in := 3, out1 => "L".MONTH)
   END_RUNG
   RUNG wire#w1
      { S7_Templates := "SrcType := USInt" } EQ_Contact(in1 := "DTL".READ.MONTH, in2 := 10)
      Move(in := 4, out1 => "L".MONTH)
   END_RUNG
   RUNG wire#w1
      { S7_Templates := "SrcType := USInt" } EQ_Contact(in1 := "DTL".READ.MONTH, in2 := 11)
      Move(in := 5, out1 => "L".MONTH)
   END_RUNG
   RUNG wire#w1
      { S7_Templates := "SrcType := USInt" } EQ_Contact(in1 := "DTL".READ.MONTH, in2 := 12)
      Move(in := 6, out1 => "L".MONTH)
   END_RUNG
   RUNG wire#w1
      { S7_Templates := "SrcType := USInt" } LT_Contact(in1 := "DTL".READ.MONTH, in2 := 7)
      Add(in1 := 6, in2 := "DTL".READ.MONTH, out => "L".MONTH)
   END_RUNG
   // the same network as SCL:
   #_w1 := NOT "AlwaysTRUE" AND ("L".MONTH = 0);
   IF #_w1 AND ("DTL".READ.MONTH = 7) THEN "L".MONTH := 1; END_IF;
   IF #_w1 AND ("DTL".READ.MONTH = 8) THEN "L".MONTH := 2; END_IF;
   IF #_w1 AND ("DTL".READ.MONTH = 9) THEN "L".MONTH := 3; END_IF;
   IF #_w1 AND ("DTL".READ.MONTH = 10) THEN "L".MONTH := 4; END_IF;
   IF #_w1 AND ("DTL".READ.MONTH = 11) THEN "L".MONTH := 5; END_IF;
   IF #_w1 AND ("DTL".READ.MONTH = 12) THEN "L".MONTH := 6; END_IF;
   IF #_w1 AND ("DTL".READ.MONTH < 7) THEN "L".MONTH := 6 + "DTL".READ.MONTH; END_IF;
END_REGION

REGION Network 9: YEAR_L
   RUNG wire#powerrail
      I_Contact( "AlwaysTRUE" )
      wire#w1
      { S7_Templates := "SrcType := USInt" } EQ_Contact(in1 := "L".MONTH, in2 := 0)
      { S7_Templates := "SrcType := USInt" } LT_Contact(in1 := "DTL".READ.MONTH, in2 := 7)
      Move(in := "DTL".READ.YEAR, out1 => "L".YEAR)
   END_RUNG
   RUNG wire#w1
      { S7_Templates := "SrcType := UInt" } EQ_Contact(in1 := "DTL".READ.YEAR, in2 := 2021)
      { S7_Templates := "SrcType := USInt" } GE_Contact(in1 := "DTL".READ.MONTH, in2 := 7)
      Add(in1 := "DTL".READ.YEAR, in2 := 1, out => "L".YEAR)
   END_RUNG
   RUNG wire#w1
      { S7_Templates := "SrcType := UInt" } EQ_Contact(in1 := "DTL".READ.YEAR, in2 := 2022)
      { S7_Templates := "SrcType := USInt" } GE_Contact(in1 := "DTL".READ.MONTH, in2 := 7)
      Add(in1 := "DTL".READ.YEAR, in2 := 1, out => "L".YEAR)
   END_RUNG
   // the same network as SCL:
   IF NOT "AlwaysTRUE" AND ("L".MONTH = 0) AND ("DTL".READ.MONTH < 7) THEN
       "L".YEAR := "DTL".READ.YEAR;
   END_IF;
   IF NOT "AlwaysTRUE" AND ("DTL".READ.YEAR = 2021) AND ("DTL".READ.MONTH >= 7) THEN
       "L".YEAR := "DTL".READ.YEAR + 1;
   END_IF;
   IF NOT "AlwaysTRUE" AND ("DTL".READ.YEAR = 2022) AND ("DTL".READ.MONTH >= 7) THEN
       "L".YEAR := "DTL".READ.YEAR + 1;
   END_IF;
END_REGION

REGION Network 10: IMP
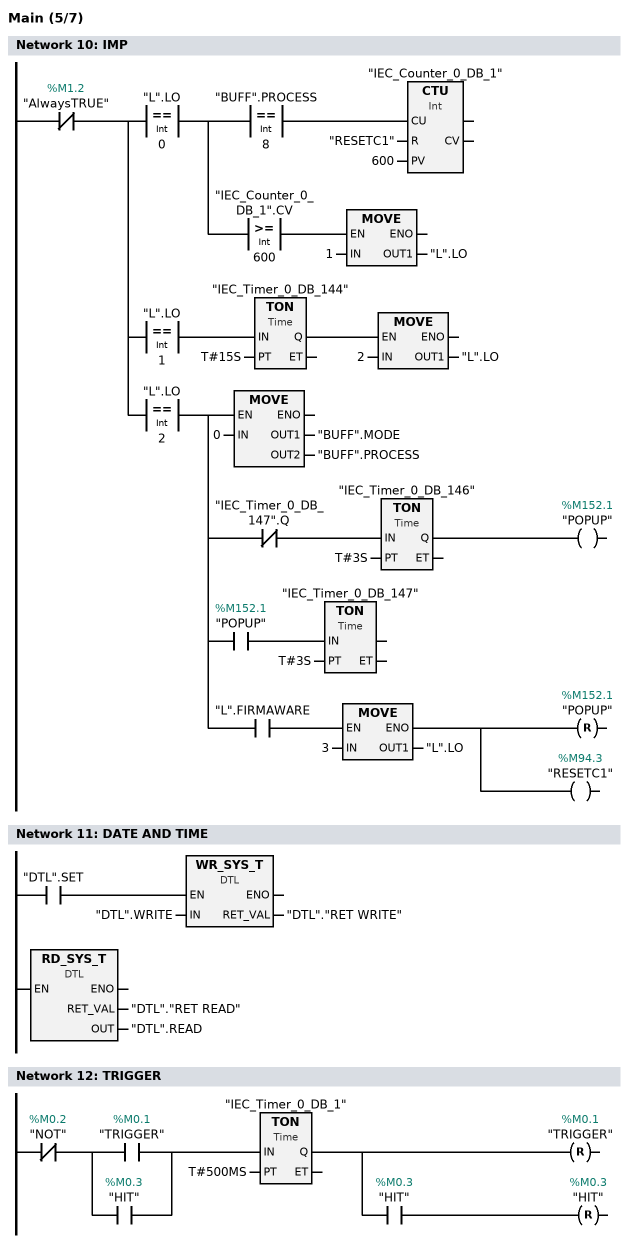
   RUNG wire#powerrail
      I_Contact( "AlwaysTRUE" )
      wire#w1
      { S7_Templates := "SrcType := Int" } EQ_Contact(in1 := "L".LO, in2 := 0)
      wire#w2
      { S7_Templates := "SrcType := Int" } EQ_Contact(in1 := "BUFF".PROCESS, in2 := 8)
      { S7_Templates := "value_type := Int" } "IEC_Counter_0_DB_1".CTU(r := "RESETC1", pv := 600, cv =>)
   END_RUNG
   RUNG wire#w2
      { S7_Templates := "SrcType := Int" } GE_Contact(in1 := "IEC_Counter_0_DB_1".CV, in2 := 600)
      Move(in := 1, out1 => "L".LO)
   END_RUNG
   RUNG wire#w1
      { S7_Templates := "SrcType := Int" } EQ_Contact(in1 := "L".LO, in2 := 1)
      { S7_Templates := "time_type := Time" } "IEC_Timer_0_DB_144".TON(pt := T#15S, et =>)
      Move(in := 2, out1 => "L".LO)
   END_RUNG
   RUNG wire#w1
      { S7_Templates := "SrcType := Int" } EQ_Contact(in1 := "L".LO, in2 := 2)
      wire#w3
      Move(in := 0, out1 => "BUFF".MODE, out2 => "BUFF".PROCESS)
   END_RUNG
   RUNG wire#w3
      I_Contact( "IEC_Timer_0_DB_147".Q )
      { S7_Templates := "time_type := Time" } "IEC_Timer_0_DB_146".TON(pt := T#3S, et =>)
      Coil( "POPUP" )
   END_RUNG
   RUNG wire#w3
      Contact( "POPUP" )
      { S7_Templates := "time_type := Time" } "IEC_Timer_0_DB_147".TON(pt := T#3S, et =>)
   END_RUNG
   RUNG wire#w3
      Contact( "L".FIRMAWARE )
      Move(in := 3, out1 => "L".LO)
      wire#w4
      R_Coil( "POPUP" )
   END_RUNG
   RUNG wire#w4
      Coil( "RESETC1" )
   END_RUNG
   // the same network as SCL:
   #_w1 := NOT "AlwaysTRUE" AND ("L".LO = 0);
   "IEC_Counter_0_DB_1".CTU(CU := #_w1 AND ("BUFF".PROCESS = 8), R := "RESETC1", PV := 600);
   IF #_w1 AND ("IEC_Counter_0_DB_1".CV >= 600) THEN "L".LO := 1; END_IF;
   "IEC_Timer_0_DB_144".TON(IN := NOT "AlwaysTRUE" AND ("L".LO = 1), PT := T#15S);
   IF "IEC_Timer_0_DB_144".Q THEN "L".LO := 2; END_IF;
   #_w2 := NOT "AlwaysTRUE" AND ("L".LO = 2);
   IF #_w2 THEN
       "BUFF".MODE := 0;
       "BUFF".PROCESS := 0;
   END_IF;
   "IEC_Timer_0_DB_146".TON(IN := #_w2 AND NOT "IEC_Timer_0_DB_147".Q, PT := T#3S);
   "POPUP" := "IEC_Timer_0_DB_146".Q;
   "IEC_Timer_0_DB_147".TON(IN := #_w2 AND "POPUP", PT := T#3S);
   #_w3 := #_w2 AND "L".FIRMAWARE;
   IF #_w3 THEN
       "L".LO := 3;
       "POPUP" := FALSE;
   END_IF;
   "RESETC1" := #_w3;
END_REGION

REGION Network 11: DATE AND TIME
   RUNG wire#powerrail
      Contact( "DTL".SET )
      { S7_Templates := "date_type := DTL" } WR_SYS_T(IN := "DTL".WRITE, RET_VAL => "DTL"."RET WRITE")
   END_RUNG
   RUNG wire#powerrail
      { S7_Templates := "date_type := DTL" } RD_SYS_T(RET_VAL => "DTL"."RET READ", OUT => "DTL".READ)
   END_RUNG
   // the same network as SCL:
   IF "DTL".SET THEN "DTL"."RET WRITE" := WR_SYS_T(IN := "DTL".WRITE); END_IF;
   "DTL"."RET READ" := RD_SYS_T(OUT => "DTL".READ);
END_REGION

REGION Network 12: TRIGGER
   RUNG wire#powerrail
      I_Contact( "NOT" )
      wire#w1
      Contact( "TRIGGER" )
      wire#w2
      { S7_Templates := "time_type := Time" } "IEC_Timer_0_DB_1".TON(pt := T#500MS, et =>)
      wire#w3
      R_Coil( "TRIGGER" )
   END_RUNG
   RUNG wire#w1
      Contact( "HIT" )
   END_RUNG wire#w2
   RUNG wire#w3
      Contact( "HIT" )
      R_Coil( "HIT" )
   END_RUNG
   // the same network as SCL:
   "IEC_Timer_0_DB_1".TON(IN := NOT "NOT" AND ("TRIGGER" OR "HIT"), PT := T#500MS);
   IF "IEC_Timer_0_DB_1".Q THEN "TRIGGER" := FALSE; END_IF;
   IF "IEC_Timer_0_DB_1".Q AND "HIT" THEN "HIT" := FALSE; END_IF;
END_REGION

REGION Network 13: CYCLE COUNT
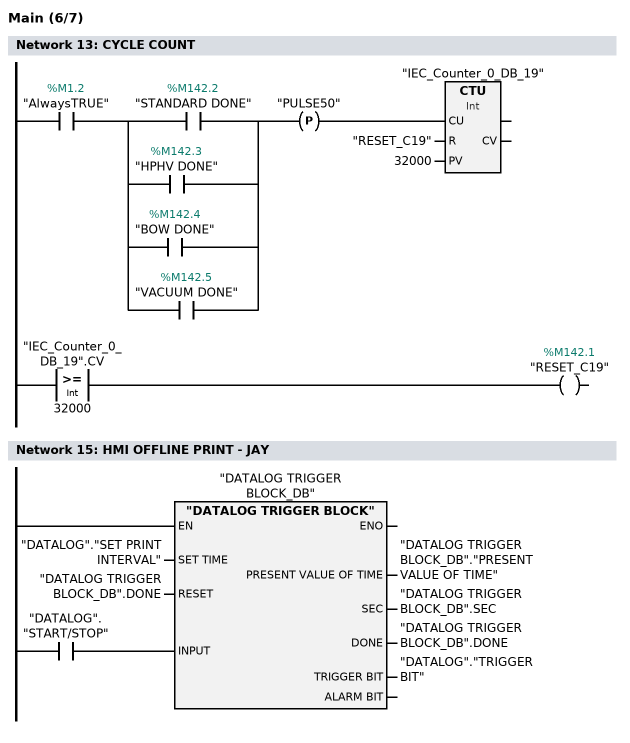
   RUNG wire#powerrail
      Contact( "AlwaysTRUE" )
      wire#w1
      Contact( "STANDARD DONE" )
      wire#w2
      P_Trig( "PULSE50" )
      { S7_Templates := "value_type := Int" } "IEC_Counter_0_DB_19".CTU(r := "RESET_C19", pv := 32000, cv =>)
   END_RUNG
   RUNG wire#w1
      Contact( "HPHV DONE" )
   END_RUNG wire#w2
   RUNG wire#w1
      Contact( "BOW DONE" )
   END_RUNG wire#w2
   RUNG wire#w1
      Contact( "VACUUM DONE" )
   END_RUNG wire#w2
   RUNG wire#powerrail
      { S7_Templates := "SrcType := Int" } GE_Contact(in1 := "IEC_Counter_0_DB_19".CV, in2 := 32000)
      Coil( "RESET_C19" )
   END_RUNG
   // the same network as SCL:
   #_w1 := "AlwaysTRUE" AND ("STANDARD DONE" OR "HPHV DONE" OR "BOW DONE" OR "VACUUM DONE");
   #_w2 := #_w1 AND NOT "PULSE50";   // rising edge
   "PULSE50" := #_w1;
   "IEC_Counter_0_DB_19".CTU(CU := #_w2, R := "RESET_C19", PV := 32000);
   "RESET_C19" := "IEC_Counter_0_DB_19".CV >= 32000;
END_REGION

REGION Network 15: HMI OFFLINE PRINT - JAY
   RUNG wire#powerrail
      "DATALOG TRIGGER BLOCK_DB"(INPUT := wire#w1, "SET TIME" := "DATALOG"."SET PRINT INTERVAL", RESET := "DATALOG TRIGGER BLOCK_DB".DONE, "PRESENT VALUE OF TIME" => "DATALOG TRIGGER BLOCK_DB"."PRESENT VALUE OF TIME", SEC => "DATALOG TRIGGER BLOCK_DB".SEC, DONE => "DATALOG TRIGGER BLOCK_DB".DONE, "TRIGGER BIT" => "DATALOG"."TRIGGER BIT", "ALARM BIT" =>)
   END_RUNG
   RUNG wire#powerrail
      Contact( "DATALOG"."START/STOP" )
   END_RUNG wire#w1
   // the same network as SCL:
   "DATALOG TRIGGER BLOCK_DB"("SET TIME" := "DATALOG"."SET PRINT INTERVAL",   // "DATALOG TRIGGER BLOCK"
                           RESET := "DATALOG TRIGGER BLOCK_DB".DONE,
                           INPUT := "DATALOG"."START/STOP",
                           "PRESENT VALUE OF TIME" => "DATALOG TRIGGER BLOCK_DB"."PRESENT VALUE OF TIME",
                           SEC => "DATALOG TRIGGER BLOCK_DB".SEC,
                           DONE => "DATALOG TRIGGER BLOCK_DB".DONE,
                           "TRIGGER BIT" => "DATALOG"."TRIGGER BIT");
END_REGION

REGION Network 16: BATCH START STOP INTERLOCK
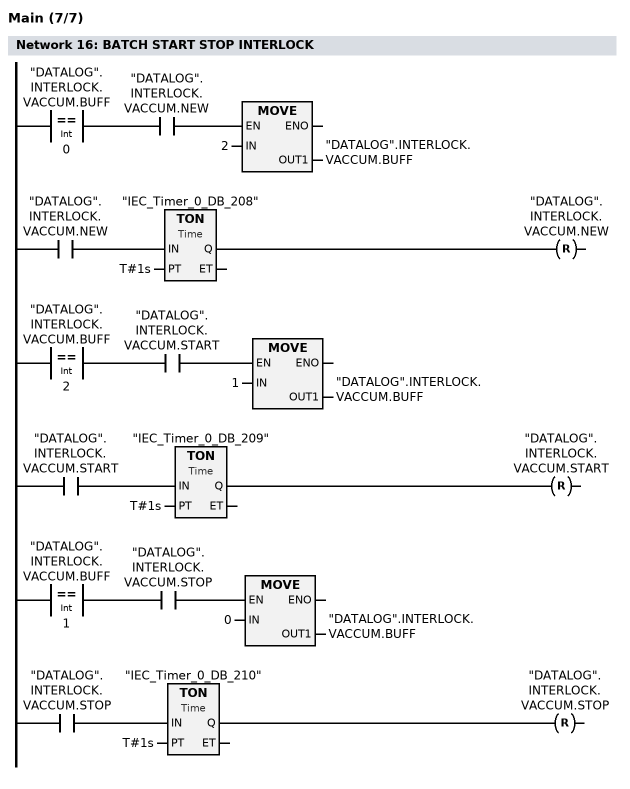
   RUNG wire#powerrail
      { S7_Templates := "SrcType := Int" } EQ_Contact(in1 := "DATALOG".INTERLOCK.VACCUM.BUFF, in2 := 0)
      Contact( "DATALOG".INTERLOCK.VACCUM.NEW )
      Move(in := 2, out1 => "DATALOG".INTERLOCK.VACCUM.BUFF)
   END_RUNG
   RUNG wire#powerrail
      Contact( "DATALOG".INTERLOCK.VACCUM.NEW )
      { S7_Templates := "time_type := Time" } "IEC_Timer_0_DB_208".TON(pt := T#1s, et =>)
      R_Coil( "DATALOG".INTERLOCK.VACCUM.NEW )
   END_RUNG
   RUNG wire#powerrail
      { S7_Templates := "SrcType := Int" } EQ_Contact(in1 := "DATALOG".INTERLOCK.VACCUM.BUFF, in2 := 2)
      Contact( "DATALOG".INTERLOCK.VACCUM.START )
      Move(in := 1, out1 => "DATALOG".INTERLOCK.VACCUM.BUFF)
   END_RUNG
   RUNG wire#powerrail
      Contact( "DATALOG".INTERLOCK.VACCUM.START )
      { S7_Templates := "time_type := Time" } "IEC_Timer_0_DB_209".TON(pt := T#1s, et =>)
      R_Coil( "DATALOG".INTERLOCK.VACCUM.START )
   END_RUNG
   RUNG wire#powerrail
      { S7_Templates := "SrcType := Int" } EQ_Contact(in1 := "DATALOG".INTERLOCK.VACCUM.BUFF, in2 := 1)
      Contact( "DATALOG".INTERLOCK.VACCUM.STOP )
      Move(in := 0, out1 => "DATALOG".INTERLOCK.VACCUM.BUFF)
   END_RUNG
   RUNG wire#powerrail
      Contact( "DATALOG".INTERLOCK.VACCUM.STOP )
      { S7_Templates := "time_type := Time" } "IEC_Timer_0_DB_210".TON(pt := T#1s, et =>)
      R_Coil( "DATALOG".INTERLOCK.VACCUM.STOP )
   END_RUNG
   // the same network as SCL:
   IF ("DATALOG".INTERLOCK.VACCUM.BUFF = 0) AND "DATALOG".INTERLOCK.VACCUM.NEW THEN
       "DATALOG".INTERLOCK.VACCUM.BUFF := 2;
   END_IF;
   "IEC_Timer_0_DB_208".TON(IN := "DATALOG".INTERLOCK.VACCUM.NEW, PT := T#1s);
   IF "IEC_Timer_0_DB_208".Q THEN "DATALOG".INTERLOCK.VACCUM.NEW := FALSE; END_IF;
   IF ("DATALOG".INTERLOCK.VACCUM.BUFF = 2) AND "DATALOG".INTERLOCK.VACCUM.START THEN
       "DATALOG".INTERLOCK.VACCUM.BUFF := 1;
   END_IF;
   "IEC_Timer_0_DB_209".TON(IN := "DATALOG".INTERLOCK.VACCUM.START, PT := T#1s);
   IF "IEC_Timer_0_DB_209".Q THEN "DATALOG".INTERLOCK.VACCUM.START := FALSE; END_IF;
   IF ("DATALOG".INTERLOCK.VACCUM.BUFF = 1) AND "DATALOG".INTERLOCK.VACCUM.STOP THEN
       "DATALOG".INTERLOCK.VACCUM.BUFF := 0;
   END_IF;
   "IEC_Timer_0_DB_210".TON(IN := "DATALOG".INTERLOCK.VACCUM.STOP, PT := T#1s);
   IF "IEC_Timer_0_DB_210".Q THEN "DATALOG".INTERLOCK.VACCUM.STOP := FALSE; END_IF;
END_REGION
END_ORGANIZATION_BLOCK

FUNCTION "PRINT PV" : Void   // FC1, LAD
{ S7_Optimized_Access := 'TRUE' }
// stored: SetENOAutomatically false
   VAR_TEMP   // added for the SCL form of the ladder/FBD networks
      _w1 : Bool;
   END_VAR
BEGIN

REGION Network 1: GET DATE AND TIME
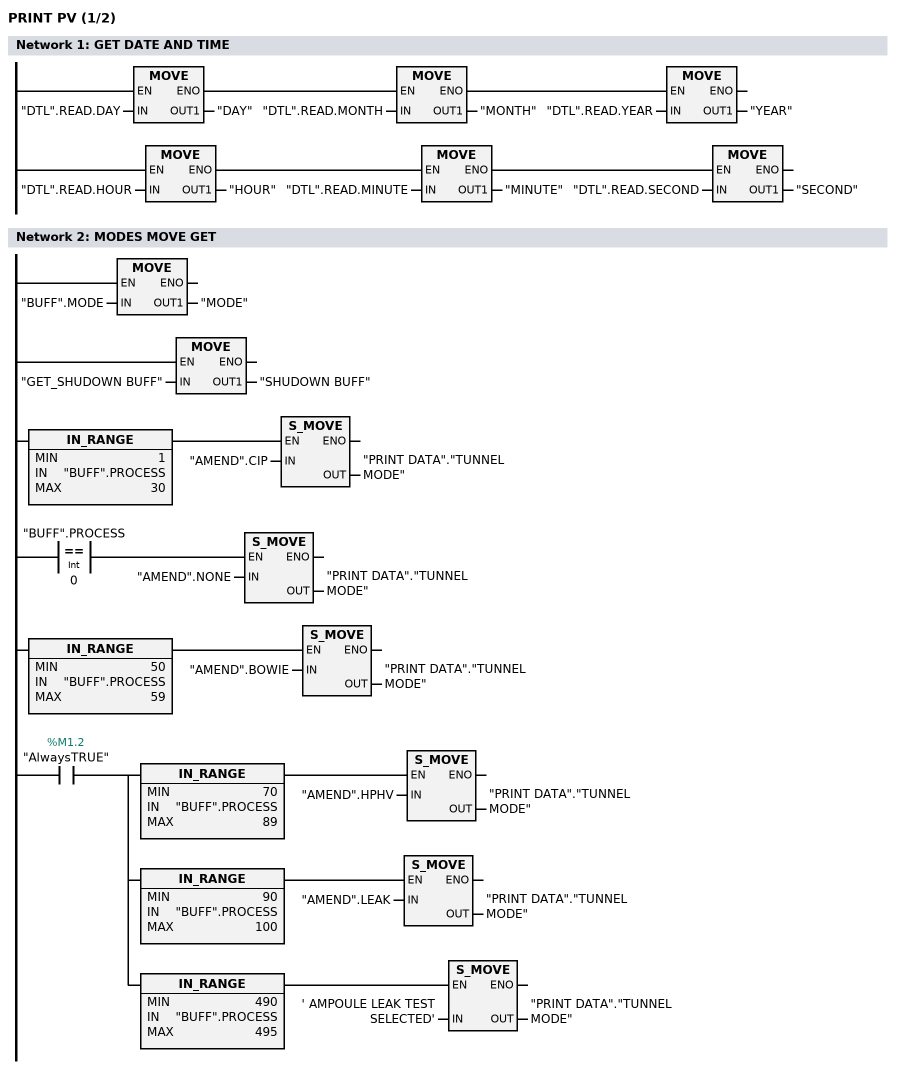
   RUNG wire#powerrail
      Move(in := "DTL".READ.DAY, out1 => "DAY")
      Move(in := "DTL".READ.MONTH, out1 => "MONTH")
      Move(in := "DTL".READ.YEAR, out1 => "YEAR")
   END_RUNG
   RUNG wire#powerrail
      Move(in := "DTL".READ.HOUR, out1 => "HOUR")
      Move(in := "DTL".READ.MINUTE, out1 => "MINUTE")
      Move(in := "DTL".READ.SECOND, out1 => "SECOND")
   END_RUNG
   // the same network as SCL:
   "DAY" := "DTL".READ.DAY;
   "MONTH" := "DTL".READ.MONTH;
   "YEAR" := "DTL".READ.YEAR;
   "HOUR" := "DTL".READ.HOUR;
   "MINUTE" := "DTL".READ.MINUTE;
   "SECOND" := "DTL".READ.SECOND;
END_REGION

REGION Network 2: MODES MOVE GET
   RUNG wire#powerrail
      Move(in := "BUFF".MODE, out1 => "MODE")
   END_RUNG
   RUNG wire#powerrail
      Move(in := "GET_SHUDOWN BUFF", out1 => "SHUDOWN BUFF")
   END_RUNG
   RUNG wire#powerrail
      { S7_Templates := "SrcType := Int" } InRange(min := 1, in := "BUFF".PROCESS, max := 30)
      S_Move(in := "AMEND".CIP, out => "PRINT DATA"."TUNNEL MODE")
   END_RUNG
   RUNG wire#powerrail
      { S7_Templates := "SrcType := Int" } EQ_Contact(in1 := "BUFF".PROCESS, in2 := 0)
      S_Move(in := "AMEND".NONE, out => "PRINT DATA"."TUNNEL MODE")
   END_RUNG
   RUNG wire#powerrail
      { S7_Templates := "SrcType := Int" } InRange(min := 50, in := "BUFF".PROCESS, max := 59)
      S_Move(in := "AMEND".BOWIE, out => "PRINT DATA"."TUNNEL MODE")
   END_RUNG
   RUNG wire#powerrail
      Contact( "AlwaysTRUE" )
      wire#w1
      { S7_Templates := "SrcType := Int" } InRange(min := 70, in := "BUFF".PROCESS, max := 89)
      S_Move(in := "AMEND".HPHV, out => "PRINT DATA"."TUNNEL MODE")
   END_RUNG
   RUNG wire#w1
      { S7_Templates := "SrcType := Int" } InRange(min := 90, in := "BUFF".PROCESS, max := 100)
      S_Move(in := "AMEND".LEAK, out => "PRINT DATA"."TUNNEL MODE")
   END_RUNG
   RUNG wire#w1
      { S7_Templates := "SrcType := Int" } InRange(min := 490, in := "BUFF".PROCESS, max := 495)
      S_Move(in := ' AMPOULE LEAK TEST SELECTED', out => "PRINT DATA"."TUNNEL MODE")
   END_RUNG
   // the same network as SCL:
   "MODE" := "BUFF".MODE;
   "SHUDOWN BUFF" := "GET_SHUDOWN BUFF";
   IF (1 <= "BUFF".PROCESS) AND ("BUFF".PROCESS <= 30) THEN
       "PRINT DATA"."TUNNEL MODE" := "AMEND".CIP;
   END_IF;
   IF "BUFF".PROCESS = 0 THEN "PRINT DATA"."TUNNEL MODE" := "AMEND".NONE; END_IF;
   IF (50 <= "BUFF".PROCESS) AND ("BUFF".PROCESS <= 59) THEN
       "PRINT DATA"."TUNNEL MODE" := "AMEND".BOWIE;
   END_IF;
   IF "AlwaysTRUE" AND (70 <= "BUFF".PROCESS) AND ("BUFF".PROCESS <= 89) THEN
       "PRINT DATA"."TUNNEL MODE" := "AMEND".HPHV;
   END_IF;
   IF "AlwaysTRUE" AND (90 <= "BUFF".PROCESS) AND ("BUFF".PROCESS <= 100) THEN
       "PRINT DATA"."TUNNEL MODE" := "AMEND".LEAK;
   END_IF;
   IF "AlwaysTRUE" AND (490 <= "BUFF".PROCESS) AND ("BUFF".PROCESS <= 495) THEN
       "PRINT DATA"."TUNNEL MODE" := ' AMPOULE LEAK TEST SELECTED';
   END_IF;
END_REGION

REGION Network 3
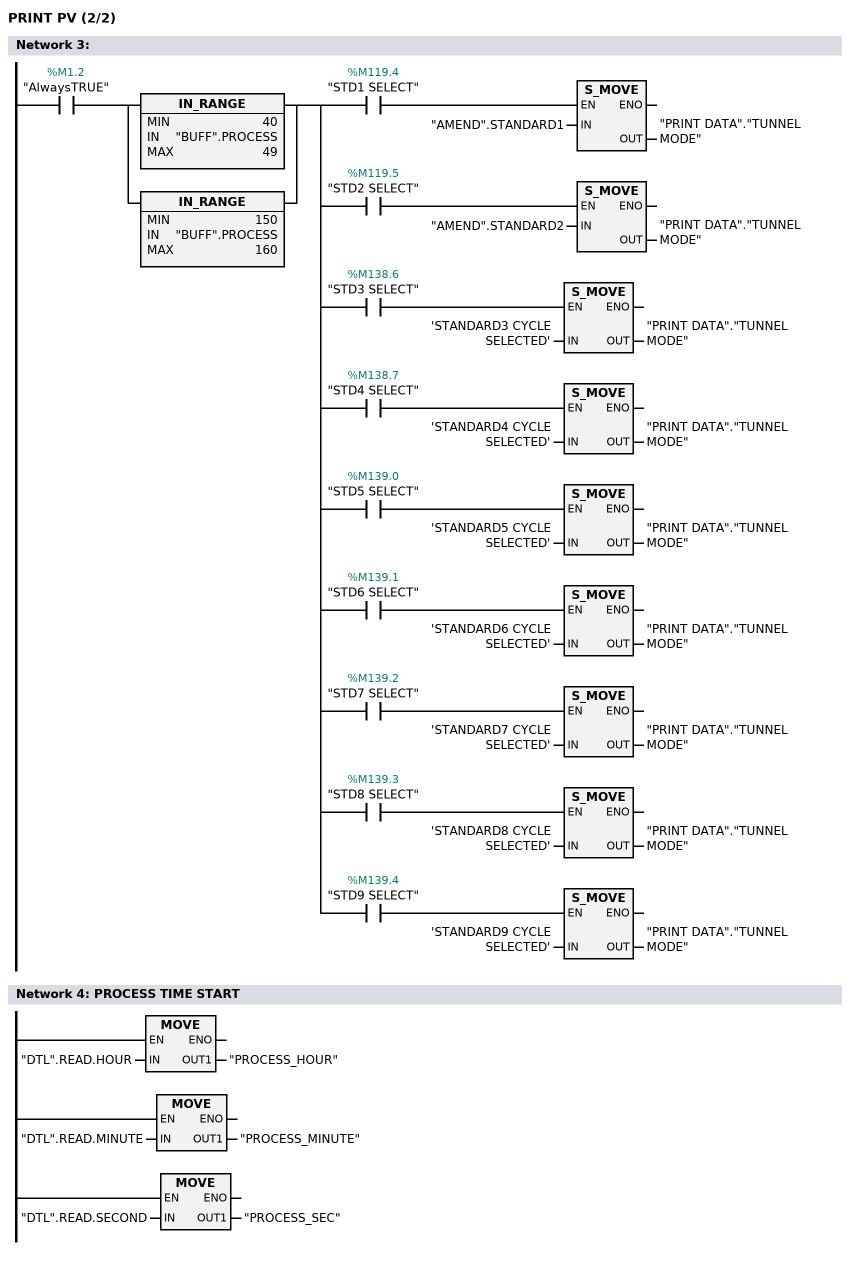
   RUNG wire#powerrail
      Contact( "AlwaysTRUE" )
      wire#w1
      { S7_Templates := "SrcType := Int" } InRange(min := 40, in := "BUFF".PROCESS, max := 49)
      wire#w2
      Contact( "STD1 SELECT" )
      S_Move(in := "AMEND".STANDARD1, out => "PRINT DATA"."TUNNEL MODE")
   END_RUNG
   RUNG wire#w1
      { S7_Templates := "SrcType := Int" } InRange(min := 150, in := "BUFF".PROCESS, max := 160)
   END_RUNG wire#w2
   RUNG wire#w2
      Contact( "STD2 SELECT" )
      S_Move(in := "AMEND".STANDARD2, out => "PRINT DATA"."TUNNEL MODE")
   END_RUNG
   RUNG wire#w2
      Contact( "STD3 SELECT" )
      S_Move(in := 'STANDARD3 CYCLE SELECTED', out => "PRINT DATA"."TUNNEL MODE")
   END_RUNG
   RUNG wire#w2
      Contact( "STD4 SELECT" )
      S_Move(in := 'STANDARD4 CYCLE SELECTED', out => "PRINT DATA"."TUNNEL MODE")
   END_RUNG
   RUNG wire#w2
      Contact( "STD5 SELECT" )
      S_Move(in := 'STANDARD5 CYCLE SELECTED', out => "PRINT DATA"."TUNNEL MODE")
   END_RUNG
   RUNG wire#w2
      Contact( "STD6 SELECT" )
      S_Move(in := 'STANDARD6 CYCLE SELECTED', out => "PRINT DATA"."TUNNEL MODE")
   END_RUNG
   RUNG wire#w2
      Contact( "STD7 SELECT" )
      S_Move(in := 'STANDARD7 CYCLE SELECTED', out => "PRINT DATA"."TUNNEL MODE")
   END_RUNG
   RUNG wire#w2
      Contact( "STD8 SELECT" )
      S_Move(in := 'STANDARD8 CYCLE SELECTED', out => "PRINT DATA"."TUNNEL MODE")
   END_RUNG
   RUNG wire#w2
      Contact( "STD9 SELECT" )
      S_Move(in := 'STANDARD9 CYCLE SELECTED', out => "PRINT DATA"."TUNNEL MODE")
   END_RUNG
   // the same network as SCL:
   #_w1 := "AlwaysTRUE" AND (((40 <= "BUFF".PROCESS) AND ("BUFF".PROCESS <= 49)) OR ((150 <= "BUFF".PROCESS) AND ("BUFF".PROCESS <= 160)));
   IF #_w1 AND "STD1 SELECT" THEN "PRINT DATA"."TUNNEL MODE" := "AMEND".STANDARD1; END_IF;
   IF #_w1 AND "STD2 SELECT" THEN "PRINT DATA"."TUNNEL MODE" := "AMEND".STANDARD2; END_IF;
   IF #_w1 AND "STD3 SELECT" THEN "PRINT DATA"."TUNNEL MODE" := 'STANDARD3 CYCLE SELECTED'; END_IF;
   IF #_w1 AND "STD4 SELECT" THEN "PRINT DATA"."TUNNEL MODE" := 'STANDARD4 CYCLE SELECTED'; END_IF;
   IF #_w1 AND "STD5 SELECT" THEN "PRINT DATA"."TUNNEL MODE" := 'STANDARD5 CYCLE SELECTED'; END_IF;
   IF #_w1 AND "STD6 SELECT" THEN "PRINT DATA"."TUNNEL MODE" := 'STANDARD6 CYCLE SELECTED'; END_IF;
   IF #_w1 AND "STD7 SELECT" THEN "PRINT DATA"."TUNNEL MODE" := 'STANDARD7 CYCLE SELECTED'; END_IF;
   IF #_w1 AND "STD8 SELECT" THEN "PRINT DATA"."TUNNEL MODE" := 'STANDARD8 CYCLE SELECTED'; END_IF;
   IF #_w1 AND "STD9 SELECT" THEN "PRINT DATA"."TUNNEL MODE" := 'STANDARD9 CYCLE SELECTED'; END_IF;
END_REGION

REGION Network 4: PROCESS TIME START
   RUNG wire#powerrail
      Move(in := "DTL".READ.HOUR, out1 => "PROCESS_HOUR")
   END_RUNG
   RUNG wire#powerrail
      Move(in := "DTL".READ.MINUTE, out1 => "PROCESS_MINUTE")
   END_RUNG
   RUNG wire#powerrail
      Move(in := "DTL".READ.SECOND, out1 => "PROCESS_SEC")
   END_RUNG
   // the same network as SCL:
   "PROCESS_HOUR" := "DTL".READ.HOUR;
   "PROCESS_MINUTE" := "DTL".READ.MINUTE;
   "PROCESS_SEC" := "DTL".READ.SECOND;
END_REGION
END_FUNCTION

FUNCTION "ALARMS PRINT" : Void   // FC2, LAD
{ S7_Optimized_Access := 'TRUE' }
// stored: SetENOAutomatically false
   VAR_TEMP   // added for the SCL form of the ladder/FBD networks
      _w1 : Bool;
      _w2 : Bool;
   END_VAR
BEGIN

REGION Network 1
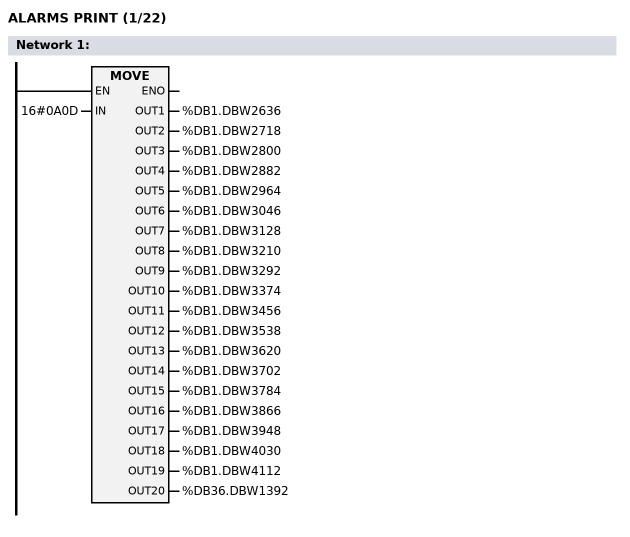
   RUNG wire#powerrail
      Move(in := 16#0A0D, out1 => %DB1.DBW2636, out2 => %DB1.DBW2718, out3 => %DB1.DBW2800, out4 => %DB1.DBW2882, out5 => %DB1.DBW2964, out6 => %DB1.DBW3046, out7 => %DB1.DBW3128, out8 => %DB1.DBW3210, out9 => %DB1.DBW3292, out10 => %DB1.DBW3374, out11 => %DB1.DBW3456, out12 => %DB1.DBW3538, out13 => %DB1.DBW3620, out14 => %DB1.DBW3702, out15 => %DB1.DBW3784, out16 => %DB1.DBW3866, out17 => %DB1.DBW3948, out18 => %DB1.DBW4030, out19 => %DB1.DBW4112, out20 => %DB36.DBW1392)
   END_RUNG
   // the same network as SCL:
   %DB1.DBW2636 := 16#0A0D;
   %DB1.DBW2718 := 16#0A0D;
   %DB1.DBW2800 := 16#0A0D;
   %DB1.DBW2882 := 16#0A0D;
   %DB1.DBW2964 := 16#0A0D;
   %DB1.DBW3046 := 16#0A0D;
   %DB1.DBW3128 := 16#0A0D;
   %DB1.DBW3210 := 16#0A0D;
   %DB1.DBW3292 := 16#0A0D;
   %DB1.DBW3374 := 16#0A0D;
   %DB1.DBW3456 := 16#0A0D;
   %DB1.DBW3538 := 16#0A0D;
   %DB1.DBW3620 := 16#0A0D;
   %DB1.DBW3702 := 16#0A0D;
   %DB1.DBW3784 := 16#0A0D;
   %DB1.DBW3866 := 16#0A0D;
   %DB1.DBW3948 := 16#0A0D;
   %DB1.DBW4030 := 16#0A0D;
   %DB1.DBW4112 := 16#0A0D;
   %DB36.DBW1392 := 16#0A0D;
END_REGION

